LIN {X -0.212,Y -498.019,Z 383.978,A 0.000,B 0.000,C 90.000,E1 212.084} C_DIS
LIN {X 0.199,Y -493.119,Z 383.966,A 0.000,B 0.000,C 90.000,E1 209.922} C_DIS
LIN {X 0.159,Y -488.917,Z 383.956,A 0.000,B 0.000,C 90.000,E1 208.103} C_DIS
LIN {X 0.025,Y -484.697,Z 383.946,A 0.000,B 0.000,C 90.000,E1 206.283} C_DIS
LIN {X -0.193,Y -481.042,Z 383.938,A 0.000,B 0.000,C 90.000,E1 204.771} C_DIS
LIN {X -0.035,Y -477.293,Z 383.929,A 0.000,B 0.000,C 90.000,E1 203.206} C_DIS
LIN {X -0.131,Y -473.559,Z 383.920,A 0.000,B 0.000,C 90.000,E1 201.663} C_DIS
LIN {X 0.100,Y -469.164,Z 383.910,A 0.000,B 0.000,C 90.000,E1 199.758} C_DIS
LIN {X -0.148,Y -464.289,Z 383.898,A 0.000,B 0.000,C 90.000,E1 197.583} C_DIS
LIN {X -0.001,Y -460.326,Z 383.887,A 0.000,B 0.000,C 90.000,E1 195.662} C_DIS
LIN {X -0.193,Y -456.648,Z 383.876,A 0.000,B 0.000,C 90.000,E1 193.772} C_DIS
LIN {X 0.206,Y -453.691,Z 383.868,A 0.000,B 0.000,C 90.000,E1 192.119} C_DIS
LIN {X -0.131,Y -449.792,Z 383.855,A 0.000,B 0.000,C 90.000,E1 189.905} C_DIS
LIN {X 0.200,Y -447.685,Z 383.848,A 0.000,B 0.000,C 90.000,E1 188.568} C_DIS
LIN {X 0.012,Y -444.252,Z 383.835,A 0.000,B 0.000,C 90.000,E1 186.315} C_DIS
LIN {X 0.167,Y -439.679,Z 383.815,A 0.000,B 0.000,C 90.000,E1 182.694} C_DIS
LIN {X 0.131,Y -435.374,Z 383.786,A 0.000,B 0.000,C 90.000,E1 177.421} C_DIS
LIN {X -0.043,Y -433.968,Z 383.766,A 0.000,B 0.000,C 90.000,E1 173.799} C_DIS
LIN {X -0.105,Y -434.156,Z 383.740,A 0.000,B 0.000,C 90.000,E1 169.162} C_DIS
LIN {X -0.121,Y -435.862,Z 383.720,A 0.000,B 0.000,C 90.000,E1 165.519} C_DIS
LIN {X 0.098,Y -439.493,Z 383.698,A 0.000,B 0.000,C 90.000,E1 161.529} C_DIS
LIN {X -0.063,Y -444.442,Z 383.676,A 0.000,B 0.000,C 90.000,E1 157.614} C_DIS
LIN {X 0.018,Y -450.294,Z 383.656,A 0.000,B 0.000,C 90.000,E1 154.024} C_DIS
LIN {X 0.167,Y -457.487,Z 383.636,A 0.000,B 0.000,C 90.000,E1 150.461} C_DIS
LIN {X 0.284,Y -467.028,Z 383.615,A 0.000,B 0.000,C 90.000,E1 146.628} C_DIS
LIN {X -0.114,Y -471.651,Z 383.606,A 0.000,B 0.000,C 90.000,E1 145.102} C_DIS
LIN {X 0.087,Y -480.605,Z 383.591,A 0.000,B 0.000,C 90.000,E1 142.271} C_DIS
LIN {X -0.050,Y -486.857,Z 383.580,A 0.000,B 0.000,C 90.000,E1 140.436} C_DIS
LIN {X -0.269,Y -492.019,Z 383.572,A 0.000,B 0.000,C 90.000,E1 138.933} C_DIS
LIN {X 0.086,Y -496.064,Z 383.565,A 0.000,B 0.000,C 90.000,E1 137.676} C_DIS
LIN {X 0.008,Y -500.717,Z 383.557,A 0.000,B 0.000,C 90.000,E1 136.176} C_DIS
LIN {X 0.010,Y -505.000,Z 383.548,A 0.000,B 0.000,C 90.000,E1 134.676} C_DIS
LIN {X -0.026,Y -507.267,Z 383.543,A 0.000,B 0.000,C 90.000,E1 133.785} C_DIS
LIN {X -0.043,Y -509.313,Z 383.538,A 0.000,B 0.000,C 90.000,E1 132.894} C_DIS
LIN {X -0.009,Y -511.116,Z 383.533,A 0.000,B 0.000,C 90.000,E1 132.000} C_DIS
LIN {X -0.330,Y -512.746,Z 383.528,A 0.000,B 0.000,C 90.000,E1 131.148} C_DIS
LIN {X -0.166,Y -513.695,Z 383.525,A 0.000,B 0.000,C 90.000,E1 130.539} C_DIS
LIN {X -0.148,Y -515.089,Z 383.519,A 0.000,B 0.000,C 90.000,E1 129.358} C_DIS
LIN {X 0.032,Y -515.562,Z 383.515,A 0.000,B 0.000,C 90.000,E1 128.749} C_DIS
LIN {X -0.175,Y -515.754,Z 383.510,A 0.000,B 0.000,C 90.000,E1 127.890} C_DIS
LIN {X -0.067,Y -515.510,Z 383.506,A 0.000,B 0.000,C 90.000,E1 126.996} C_DIS
LIN {X 0.141,Y -514.805,Z 383.501,A 0.000,B 0.000,C 90.000,E1 126.091} C_DIS
LIN {X -0.002,Y -514.194,Z 383.497,A 0.000,B 0.000,C 90.000,E1 125.518} C_DIS
LIN {X 0.195,Y -512.974,Z 383.492,A 0.000,B 0.000,C 90.000,E1 124.612} C_DIS
LIN {X 0.035,Y -511.972,Z 383.489,A 0.000,B 0.000,C 90.000,E1 124.040} C_DIS
LIN {X -0.079,Y -510.194,Z 383.484,A 0.000,B 0.000,C 90.000,E1 123.166} C_DIS
LIN {X 0.125,Y -507.190,Z 383.478,A 0.000,B 0.000,C 90.000,E1 121.957} C_DIS
LIN {X -0.089,Y -505.513,Z 383.474,A 0.000,B 0.000,C 90.000,E1 121.386} C_DIS
LIN {X 0.164,Y -502.742,Z 383.469,A 0.000,B 0.000,C 90.000,E1 120.463} C_DIS
LIN {X -0.048,Y -499.626,Z 383.464,A 0.000,B 0.000,C 90.000,E1 119.589} C_DIS
LIN {X 0.174,Y -495.038,Z 383.458,A 0.000,B 0.000,C 90.000,E1 118.359} C_DIS
LIN {X -0.135,Y -490.540,Z 383.452,A 0.000,B 0.000,C 90.000,E1 117.334} C_DIS
LIN {X 0.156,Y -485.837,Z 383.446,A 0.000,B 0.000,C 90.000,E1 116.232} C_DIS
LIN {X -0.051,Y -481.546,Z 383.441,A 0.000,B 0.000,C 90.000,E1 115.335} C_DIS
LIN {X -0.121,Y -474.894,Z 383.433,A 0.000,B 0.000,C 90.000,E1 113.951} C_DIS
LIN {X 0.127,Y -467.905,Z 383.425,A 0.000,B 0.000,C 90.000,E1 112.514} C_DIS
LIN {X 0.070,Y -460.775,Z 383.417,A 0.000,B 0.000,C 90.000,E1 111.099} C_DIS
LIN {X 0.102,Y -456.211,Z 383.412,A 0.000,B 0.000,C 90.000,E1 110.174} C_DIS
LIN {X 0.063,Y -456.211,Z 383.412,A 0.000,B 0.000,C 90.000,E1 110.174} C_DIS
LIN {X -0.106,Y -457.519,Z 383.409,A 0.000,B 0.000,C 90.000,E1 109.685} C_DIS
LIN {X -0.161,Y -466.202,Z 383.386,A 0.000,B 0.000,C 90.000,E1 105.552} C_DIS
LIN {X 0.015,Y -467.767,Z 383.383,A 0.000,B 0.000,C 90.000,E1 104.898} C_DIS
LIN {X -0.013,Y -475.973,Z 383.357,A 0.000,B 0.000,C 90.000,E1 100.197} C_DIS
LIN {X 0.136,Y -476.681,Z 383.353,A 0.000,B 0.000,C 90.000,E1 99.557} C_DIS
LIN {X -0.218,Y -481.919,Z 383.331,A 0.000,B 0.000,C 90.000,E1 95.568} C_DIS
LIN {X 0.109,Y -482.204,Z 383.329,A 0.000,B 0.000,C 90.000,E1 95.220} C_DIS
LIN {X 0.048,Y -485.393,Z 383.305,A 0.000,B 0.000,C 90.000,E1 90.917} C_DIS
LIN {X -0.128,Y -485.529,Z 383.303,A 0.000,B 0.000,C 90.000,E1 90.630} C_DIS
LIN {X 0.080,Y -486.360,Z 383.281,A 0.000,B 0.000,C 90.000,E1 86.617} C_DIS
LIN {X -0.095,Y -486.368,Z 383.280,A 0.000,B 0.000,C 90.000,E1 86.331} C_DIS
LIN {X -0.106,Y -485.856,Z 383.275,A 0.000,B 0.000,C 90.000,E1 85.412} C_DIS
LIN {X -0.071,Y -484.692,Z 383.254,A 0.000,B 0.000,C 90.000,E1 81.724} C_DIS
LIN {X -0.203,Y -484.502,Z 383.252,A 0.000,B 0.000,C 90.000,E1 81.432} C_DIS
LIN {X 0.134,Y -480.434,Z 383.227,A 0.000,B 0.000,C 90.000,E1 76.769} C_DIS
LIN {X -0.225,Y -474.000,Z 383.200,A 0.000,B 0.000,C 90.000,E1 72.000} C_DIS
LIN {X 0.185,Y -473.730,Z 383.199,A 0.000,B 0.000,C 90.000,E1 71.819} C_DIS
LIN {X 0.144,Y -473.739,Z 383.199,A 0.000,B 0.000,C 90.000,E1 71.819} C_DIS
LIN {X 0.186,Y -482.818,Z 383.192,A 0.000,B 0.000,C 90.000,E1 70.550} C_DIS
LIN {X -0.179,Y -490.319,Z 383.186,A 0.000,B 0.000,C 90.000,E1 69.518} C_DIS
LIN {X -0.073,Y -496.699,Z 383.181,A 0.000,B 0.000,C 90.000,E1 68.592} C_DIS
LIN {X 0.110,Y -502.654,Z 383.176,A 0.000,B 0.000,C 90.000,E1 67.667} C_DIS
LIN {X 0.006,Y -510.529,Z 383.169,A 0.000,B 0.000,C 90.000,E1 66.357} C_DIS
LIN {X -0.302,Y -515.869,Z 383.163,A 0.000,B 0.000,C 90.000,E1 65.357} C_DIS
LIN {X -0.131,Y -517.950,Z 383.160,A 0.000,B 0.000,C 90.000,E1 64.897} C_DIS
LIN {X 0.171,Y -518.682,Z 383.160,A 0.000,B 0.000,C 90.000,E1 64.717} C_DIS
LIN {X 0.140,Y -520.608,Z 383.157,A 0.000,B 0.000,C 90.000,E1 64.280} C_DIS
LIN {X -0.189,Y -521.866,Z 383.156,A 0.000,B 0.000,C 90.000,E1 64.024} C_DIS
LIN {X -0.132,Y -524.336,Z 383.152,A 0.000,B 0.000,C 90.000,E1 63.435} C_DIS
LIN {X -0.294,Y -526.545,Z 383.149,A 0.000,B 0.000,C 90.000,E1 62.871} C_DIS
LIN {X -0.094,Y -530.547,Z 383.143,A 0.000,B 0.000,C 90.000,E1 61.691} C_DIS
LIN {X 0.205,Y -533.162,Z 383.138,A 0.000,B 0.000,C 90.000,E1 60.795} C_DIS
LIN {X 0.059,Y -535.621,Z 383.133,A 0.000,B 0.000,C 90.000,E1 59.950} C_DIS
LIN {X 0.204,Y -538.712,Z 383.127,A 0.000,B 0.000,C 90.000,E1 58.791} C_DIS
LIN {X 0.118,Y -541.438,Z 383.120,A 0.000,B 0.000,C 90.000,E1 57.661} C_DIS
LIN {X -0.098,Y -543.793,Z 383.114,A 0.000,B 0.000,C 90.000,E1 56.548} C_DIS
LIN {X 0.141,Y -545.326,Z 383.109,A 0.000,B 0.000,C 90.000,E1 55.674} C_DIS
LIN {X 0.213,Y -546.196,Z 383.106,A 0.000,B 0.000,C 90.000,E1 55.102} C_DIS
LIN {X -0.021,Y -546.950,Z 383.103,A 0.000,B 0.000,C 90.000,E1 54.562} C_DIS
LIN {X 0.111,Y -547.808,Z 383.098,A 0.000,B 0.000,C 90.000,E1 53.703} C_DIS
LIN {X 0.304,Y -548.476,Z 383.092,A 0.000,B 0.000,C 90.000,E1 52.557} C_DIS
LIN {X -0.029,Y -548.669,Z 383.089,A 0.000,B 0.000,C 90.000,E1 52.029} C_DIS
LIN {X 0.072,Y -548.643,Z 383.086,A 0.000,B 0.000,C 90.000,E1 51.457} C_DIS
LIN {X -0.205,Y -548.446,Z 383.081,A 0.000,B 0.000,C 90.000,E1 50.642} C_DIS
LIN {X 0.332,Y -547.697,Z 383.075,A 0.000,B 0.000,C 90.000,E1 49.461} C_DIS
LIN {X 0.039,Y -546.848,Z 383.070,A 0.000,B 0.000,C 90.000,E1 48.647} C_DIS
LIN {X -0.280,Y -545.318,Z 383.064,A 0.000,B 0.000,C 90.000,E1 47.553} C_DIS
LIN {X 0.165,Y -542.833,Z 383.055,A 0.000,B 0.000,C 90.000,E1 45.810} C_DIS
LIN {X 0.167,Y -540.290,Z 383.045,A 0.000,B 0.000,C 90.000,E1 44.109} C_DIS
LIN {X 0.100,Y -537.579,Z 383.034,A 0.000,B 0.000,C 90.000,E1 42.123} C_DIS
LIN {X -0.007,Y -534.998,Z 383.023,A 0.000,B 0.000,C 90.000,E1 40.135} C_DIS
LIN {X 0.300,Y -532.441,Z 383.012,A 0.000,B 0.000,C 90.000,E1 38.096} C_DIS
LIN {X 0.253,Y -530.574,Z 383.004,A 0.000,B 0.000,C 90.000,E1 36.664} C_DIS
LIN {X 0.149,Y -528.249,Z 382.994,A 0.000,B 0.000,C 90.000,E1 34.945} C_DIS
LIN {X 0.148,Y -526.357,Z 382.986,A 0.000,B 0.000,C 90.000,E1 33.499} C_DIS
LIN {X 0.187,Y -523.741,Z 382.975,A 0.000,B 0.000,C 90.000,E1 31.465} C_DIS
LIN {X 0.012,Y -520.809,Z 382.962,A 0.000,B 0.000,C 90.000,E1 29.155} C_DIS
LIN {X 0.165,Y -518.751,Z 382.952,A 0.000,B 0.000,C 90.000,E1 27.385} C_DIS
LIN {X 0.150,Y -516.488,Z 382.941,A 0.000,B 0.000,C 90.000,E1 25.335} C_DIS
LIN {X 0.115,Y -514.395,Z 382.929,A 0.000,B 0.000,C 90.000,E1 23.281} C_DIS
LIN {X -0.092,Y -511.838,Z 382.913,A 0.000,B 0.000,C 90.000,E1 20.355} C_DIS
LIN {X -0.094,Y -510.019,Z 382.898,A 0.000,B 0.000,C 90.000,E1 17.692} C_DIS
LIN {X -0.007,Y -508.836,Z 382.887,A 0.000,B 0.000,C 90.000,E1 15.607} C_DIS
LIN {X -0.052,Y -507.801,Z 382.872,A 0.000,B 0.000,C 90.000,E1 12.939} C_DIS
LIN {X -0.022,Y -507.332,Z 382.855,A 0.000,B 0.000,C 90.000,E1 9.962} C_DIS
LIN {X -0.122,Y -507.550,Z 382.841,A 0.000,B 0.000,C 90.000,E1 7.296} C_DIS
LIN {X -0.001,Y -508.745,Z 382.822,A 0.000,B 0.000,C 90.000,E1 4.012} C_DIS
LIN {X -0.043,Y -511.351,Z 382.803,A 0.000,B 0.000,C 90.000,E1 0.458} C_DIS
LIN {X -0.032,Y -515.651,Z 382.783,A 0.000,B 0.000,C 90.000,E1 356.846} C_DIS
LIN {X -0.032,Y -519.661,Z 382.768,A 0.000,B 0.000,C 90.000,E1 354.204} C_DIS
LIN {X -0.271,Y -523.319,Z 382.756,A 0.000,B 0.000,C 90.000,E1 352.186} C_DIS
LIN {X -0.151,Y -532.010,Z 382.734,A 0.000,B 0.000,C 90.000,E1 348.117} C_DIS
LIN {X 0.081,Y -539.526,Z 382.718,A 0.000,B 0.000,C 90.000,E1 345.227} C_DIS
LIN {X -0.263,Y -544.311,Z 382.709,A 0.000,B 0.000,C 90.000,E1 343.559} C_DIS
LIN {X 0.123,Y -546.738,Z 382.704,A 0.000,B 0.000,C 90.000,E1 342.670} C_DIS
LIN {X 0.000,Y -550.798,Z 382.696,A 0.000,B 0.000,C 90.000,E1 341.275} C_DIS
LIN {X -0.048,Y -554.954,Z 382.688,A 0.000,B 0.000,C 90.000,E1 339.880} C_DIS
LIN {X 0.172,Y -559.088,Z 382.681,A 0.000,B 0.000,C 90.000,E1 338.465} C_DIS
LIN {X -0.050,Y -563.189,Z 382.673,A 0.000,B 0.000,C 90.000,E1 337.102} C_DIS
LIN {X 0.123,Y -568.179,Z 382.664,A 0.000,B 0.000,C 90.000,E1 335.433} C_DIS
LIN {X -0.157,Y -573.249,Z 382.655,A 0.000,B 0.000,C 90.000,E1 333.819} C_DIS
LIN {X -0.235,Y -581.148,Z 382.641,A 0.000,B 0.000,C 90.000,E1 331.385} C_DIS
LIN {X 0.090,Y -588.403,Z 382.629,A 0.000,B 0.000,C 90.000,E1 329.203} C_DIS
LIN {X 0.117,Y -592.882,Z 382.622,A 0.000,B 0.000,C 90.000,E1 327.867} C_DIS
LIN {X 0.167,Y -599.167,Z 382.611,A 0.000,B 0.000,C 90.000,E1 326.008} C_DIS
LIN {X -0.125,Y -605.669,Z 382.601,A 0.000,B 0.000,C 90.000,E1 324.196} C_DIS
LIN {X 0.085,Y -612.260,Z 382.591,A 0.000,B 0.000,C 90.000,E1 322.351} C_DIS
LIN {X -0.271,Y -617.075,Z 382.584,A 0.000,B 0.000,C 90.000,E1 321.090} C_DIS
LIN {X -0.222,Y -622.892,Z 382.575,A 0.000,B 0.000,C 90.000,E1 319.542} C_DIS
LIN {X -0.127,Y -628.524,Z 382.567,A 0.000,B 0.000,C 90.000,E1 318.000} C_DIS
LIN {X -0.151,Y -632.208,Z 382.561,A 0.000,B 0.000,C 90.000,E1 316.986} C_DIS
LIN {X -0.126,Y -635.898,Z 382.555,A 0.000,B 0.000,C 90.000,E1 315.972} C_DIS
LIN {X 0.050,Y -643.196,Z 382.544,A 0.000,B 0.000,C 90.000,E1 313.947} C_DIS
LIN {X 0.090,Y -648.799,Z 382.536,A 0.000,B 0.000,C 90.000,E1 312.447} C_DIS
LIN {X 0.244,Y -655.166,Z 382.526,A 0.000,B 0.000,C 90.000,E1 310.701} C_DIS
LIN {X 0.125,Y -661.283,Z 382.517,A 0.000,B 0.000,C 90.000,E1 308.991} C_DIS
LIN {X 0.158,Y -666.149,Z 382.509,A 0.000,B 0.000,C 90.000,E1 307.523} C_DIS
LIN {X -0.219,Y -669.305,Z 382.503,A 0.000,B 0.000,C 90.000,E1 306.583} C_DIS
LIN {X -0.041,Y -673.071,Z 382.496,A 0.000,B 0.000,C 90.000,E1 305.358} C_DIS
LIN {X -0.043,Y -677.288,Z 382.488,A 0.000,B 0.000,C 90.000,E1 303.913} C_DIS
LIN {X -0.120,Y -679.965,Z 382.483,A 0.000,B 0.000,C 90.000,E1 302.959} C_DIS
LIN {X 0.226,Y -681.866,Z 382.479,A 0.000,B 0.000,C 90.000,E1 302.212} C_DIS
LIN {X -0.174,Y -684.909,Z 382.472,A 0.000,B 0.000,C 90.000,E1 301.052} C_DIS
LIN {X 0.244,Y -686.100,Z 382.470,A 0.000,B 0.000,C 90.000,E1 300.541} C_DIS
LIN {X -0.292,Y -687.664,Z 382.466,A 0.000,B 0.000,C 90.000,E1 299.873} C_DIS
LIN {X -0.219,Y -688.947,Z 382.462,A 0.000,B 0.000,C 90.000,E1 299.155} C_DIS
LIN {X -0.270,Y -690.464,Z 382.455,A 0.000,B 0.000,C 90.000,E1 297.975} C_DIS
LIN {X -0.170,Y -690.972,Z 382.451,A 0.000,B 0.000,C 90.000,E1 297.257} C_DIS
LIN {X -0.071,Y -691.259,Z 382.447,A 0.000,B 0.000,C 90.000,E1 296.539} C_DIS
LIN {X -0.278,Y -691.343,Z 382.444,A 0.000,B 0.000,C 90.000,E1 295.848} C_DIS
LIN {X -0.037,Y -691.243,Z 382.442,A 0.000,B 0.000,C 90.000,E1 295.591} C_DIS
LIN {X 0.202,Y -691.331,Z 382.441,A 0.000,B 0.000,C 90.000,E1 295.335} C_DIS
LIN {X -0.239,Y -691.030,Z 382.438,A 0.000,B 0.000,C 90.000,E1 294.899} C_DIS
LIN {X 0.190,Y -690.803,Z 382.434,A 0.000,B 0.000,C 90.000,E1 294.155} C_DIS
LIN {X -0.012,Y -690.231,Z 382.430,A 0.000,B 0.000,C 90.000,E1 293.462} C_DIS
LIN {X -0.223,Y -689.463,Z 382.426,A 0.000,B 0.000,C 90.000,E1 292.770} C_DIS
LIN {X 0.192,Y -688.369,Z 382.422,A 0.000,B 0.000,C 90.000,E1 292.025} C_DIS
LIN {X 0.092,Y -685.866,Z 382.415,A 0.000,B 0.000,C 90.000,E1 290.610} C_DIS
LIN {X -0.106,Y -682.586,Z 382.405,A 0.000,B 0.000,C 90.000,E1 288.960} C_DIS
LIN {X -0.081,Y -680.099,Z 382.399,A 0.000,B 0.000,C 90.000,E1 287.764} C_DIS
LIN {X -0.041,Y -678.147,Z 382.393,A 0.000,B 0.000,C 90.000,E1 286.804} C_DIS
LIN {X -0.179,Y -674.689,Z 382.384,A 0.000,B 0.000,C 90.000,E1 285.134} C_DIS
LIN {X -0.234,Y -669.113,Z 382.368,A 0.000,B 0.000,C 90.000,E1 282.243} C_DIS
LIN {X -0.046,Y -664.999,Z 382.353,A 0.000,B 0.000,C 90.000,E1 279.557} C_DIS
LIN {X -0.196,Y -660.985,Z 382.333,A 0.000,B 0.000,C 90.000,E1 275.910} C_DIS
LIN {X -0.128,Y -659.346,Z 382.318,A 0.000,B 0.000,C 90.000,E1 273.212} C_DIS
LIN {X 0.049,Y -658.757,Z 382.304,A 0.000,B 0.000,C 90.000,E1 270.745} C_DIS
LIN {X 0.073,Y -658.628,Z 382.295,A 0.000,B 0.000,C 90.000,E1 269.026} C_DIS
LIN {X 0.172,Y -658.705,Z 382.291,A 0.000,B 0.000,C 90.000,E1 268.282} C_DIS
LIN {X 0.047,Y -658.927,Z 382.280,A 0.000,B 0.000,C 90.000,E1 266.331} C_DIS
LIN {X 0.312,Y -659.082,Z 382.272,A 0.000,B 0.000,C 90.000,E1 264.837} C_DIS
LIN {X -0.212,Y -659.061,Z 382.267,A 0.000,B 0.000,C 90.000,E1 264.147} C_DIS
LIN {X -0.011,Y -658.779,Z 382.263,A 0.000,B 0.000,C 90.000,E1 263.394} C_DIS
LIN {X 0.112,Y -658.258,Z 382.259,A 0.000,B 0.000,C 90.000,E1 262.648} C_DIS
LIN {X 0.311,Y -657.608,Z 382.255,A 0.000,B 0.000,C 90.000,E1 261.894} C_DIS
LIN {X -0.145,Y -656.638,Z 382.251,A 0.000,B 0.000,C 90.000,E1 261.197} C_DIS
LIN {X -0.366,Y -656.173,Z 382.250,A 0.000,B 0.000,C 90.000,E1 260.971} C_DIS
LIN {X 0.041,Y -655.553,Z 382.247,A 0.000,B 0.000,C 90.000,E1 260.443} C_DIS
LIN {X 0.213,Y -654.345,Z 382.243,A 0.000,B 0.000,C 90.000,E1 259.690} C_DIS
LIN {X -0.275,Y -653.063,Z 382.239,A 0.000,B 0.000,C 90.000,E1 258.993} C_DIS
LIN {X -0.135,Y -651.333,Z 382.233,A 0.000,B 0.000,C 90.000,E1 257.993} C_DIS
LIN {X -0.008,Y -649.355,Z 382.228,A 0.000,B 0.000,C 90.000,E1 256.992} C_DIS
LIN {X 0.227,Y -647.739,Z 382.224,A 0.000,B 0.000,C 90.000,E1 256.228} C_DIS
LIN {X 0.301,Y -645.198,Z 382.218,A 0.000,B 0.000,C 90.000,E1 255.227} C_DIS
LIN {X -0.115,Y -642.407,Z 382.213,A 0.000,B 0.000,C 90.000,E1 254.267} C_DIS
LIN {X -0.103,Y -638.482,Z 382.206,A 0.000,B 0.000,C 90.000,E1 253.015} C_DIS
LIN {X -0.170,Y -634.126,Z 382.199,A 0.000,B 0.000,C 90.000,E1 251.764} C_DIS
LIN {X 0.078,Y -630.416,Z 382.193,A 0.000,B 0.000,C 90.000,E1 250.732} C_DIS
LIN {X 0.278,Y -625.534,Z 382.186,A 0.000,B 0.000,C 90.000,E1 249.444} C_DIS
LIN {X -0.174,Y -621.492,Z 382.180,A 0.000,B 0.000,C 90.000,E1 248.465} C_DIS
LIN {X -0.150,Y -615.178,Z 382.172,A 0.000,B 0.000,C 90.000,E1 246.922} C_DIS
LIN {X -0.062,Y -607.557,Z 382.162,A 0.000,B 0.000,C 90.000,E1 245.101} C_DIS
LIN {X 0.164,Y -600.939,Z 382.153,A 0.000,B 0.000,C 90.000,E1 243.512} C_DIS
LIN {X -0.287,Y -594.283,Z 382.144,A 0.000,B 0.000,C 90.000,E1 241.975} C_DIS
LIN {X 0.317,Y -588.841,Z 382.137,A 0.000,B 0.000,C 90.000,E1 240.589} C_DIS
LIN {X 0.217,Y -580.434,Z 382.125,A 0.000,B 0.000,C 90.000,E1 238.456} C_DIS
LIN {X 0.189,Y -572.528,Z 382.113,A 0.000,B 0.000,C 90.000,E1 236.294} C_DIS
LIN {X 0.220,Y -564.219,Z 382.099,A 0.000,B 0.000,C 90.000,E1 233.829} C_DIS
LIN {X -0.039,Y -559.593,Z 382.092,A 0.000,B 0.000,C 90.000,E1 232.477} C_DIS
LIN {X -0.039,Y -554.849,Z 382.084,A 0.000,B 0.000,C 90.000,E1 231.090} C_DIS
LIN {X 0.002,Y -546.340,Z 382.070,A 0.000,B 0.000,C 90.000,E1 228.566} C_DIS
LIN {X 0.061,Y -539.958,Z 382.059,A 0.000,B 0.000,C 90.000,E1 226.581} C_DIS
LIN {X -0.006,Y -534.551,Z 382.049,A 0.000,B 0.000,C 90.000,E1 224.879} C_DIS
LIN {X -0.157,Y -530.139,Z 382.041,A 0.000,B 0.000,C 90.000,E1 223.461} C_DIS
LIN {X 0.319,Y -524.906,Z 382.032,A 0.000,B 0.000,C 90.000,E1 221.676} C_DIS
LIN {X 0.272,Y -519.007,Z 382.020,A 0.000,B 0.000,C 90.000,E1 219.644} C_DIS
LIN {X 0.154,Y -513.317,Z 382.009,A 0.000,B 0.000,C 90.000,E1 217.604} C_DIS
LIN {X 0.202,Y -507.081,Z 381.996,A 0.000,B 0.000,C 90.000,E1 215.231} C_DIS
LIN {X 0.125,Y -502.630,Z 381.986,A 0.000,B 0.000,C 90.000,E1 213.452} C_DIS
LIN {X -0.044,Y -498.327,Z 381.976,A 0.000,B 0.000,C 90.000,E1 211.671} C_DIS
LIN {X -0.147,Y -494.179,Z 381.966,A 0.000,B 0.000,C 90.000,E1 209.873} C_DIS
LIN {X -0.173,Y -490.686,Z 381.957,A 0.000,B 0.000,C 90.000,E1 208.359} C_DIS
LIN {X -0.253,Y -485.788,Z 381.946,A 0.000,B 0.000,C 90.000,E1 206.232} C_DIS
LIN {X 0.197,Y -482.142,Z 381.937,A 0.000,B 0.000,C 90.000,E1 204.643} C_DIS
LIN {X -0.068,Y -478.405,Z 381.928,A 0.000,B 0.000,C 90.000,E1 203.131} C_DIS
LIN {X -0.129,Y -475.457,Z 381.922,A 0.000,B 0.000,C 90.000,E1 201.897} C_DIS
LIN {X -0.061,Y -470.317,Z 381.909,A 0.000,B 0.000,C 90.000,E1 199.704} C_DIS
LIN {X -0.067,Y -466.143,Z 381.899,A 0.000,B 0.000,C 90.000,E1 197.819} C_DIS
LIN {X -0.091,Y -461.496,Z 381.887,A 0.000,B 0.000,C 90.000,E1 195.607} C_DIS
LIN {X -0.035,Y -458.433,Z 381.878,A 0.000,B 0.000,C 90.000,E1 194.008} C_DIS
LIN {X -0.044,Y -455.447,Z 381.869,A 0.000,B 0.000,C 90.000,E1 192.411} C_DIS
LIN {X -0.129,Y -450.955,Z 381.855,A 0.000,B 0.000,C 90.000,E1 189.849} C_DIS
LIN {X 0.222,Y -448.835,Z 381.848,A 0.000,B 0.000,C 90.000,E1 188.511} C_DIS
LIN {X 0.067,Y -445.397,Z 381.835,A 0.000,B 0.000,C 90.000,E1 186.258} C_DIS
LIN {X -0.167,Y -440.791,Z 381.815,A 0.000,B 0.000,C 90.000,E1 182.694} C_DIS
LIN {X 0.101,Y -436.798,Z 381.789,A 0.000,B 0.000,C 90.000,E1 178.051} C_DIS
LIN {X -0.032,Y -435.628,Z 381.776,A 0.000,B 0.000,C 90.000,E1 175.755} C_DIS
LIN {X -0.129,Y -434.933,Z 381.764,A 0.000,B 0.000,C 90.000,E1 173.451} C_DIS
LIN {X 0.035,Y -435.111,Z 381.741,A 0.000,B 0.000,C 90.000,E1 169.454} C_DIS
LIN {X 0.189,Y -436.902,Z 381.719,A 0.000,B 0.000,C 90.000,E1 165.463} C_DIS
LIN {X 0.032,Y -440.529,Z 381.697,A 0.000,B 0.000,C 90.000,E1 161.529} C_DIS
LIN {X 0.229,Y -446.435,Z 381.672,A 0.000,B 0.000,C 90.000,E1 156.922} C_DIS
LIN {X -0.079,Y -451.905,Z 381.654,A 0.000,B 0.000,C 90.000,E1 153.717} C_DIS
LIN {X -0.273,Y -459.246,Z 381.634,A 0.000,B 0.000,C 90.000,E1 150.205} C_DIS
LIN {X -0.091,Y -469.012,Z 381.613,A 0.000,B 0.000,C 90.000,E1 146.373} C_DIS
LIN {X 0.195,Y -473.660,Z 381.604,A 0.000,B 0.000,C 90.000,E1 144.769} C_DIS
LIN {X -0.109,Y -481.755,Z 381.591,A 0.000,B 0.000,C 90.000,E1 142.316} C_DIS
LIN {X 0.164,Y -487.989,Z 381.580,A 0.000,B 0.000,C 90.000,E1 140.436} C_DIS
LIN {X -0.032,Y -493.150,Z 381.572,A 0.000,B 0.000,C 90.000,E1 138.933} C_DIS
LIN {X 0.007,Y -497.187,Z 381.565,A 0.000,B 0.000,C 90.000,E1 137.715} C_DIS
LIN {X -0.061,Y -501.831,Z 381.557,A 0.000,B 0.000,C 90.000,E1 136.215} C_DIS
LIN {X -0.047,Y -506.093,Z 381.548,A 0.000,B 0.000,C 90.000,E1 134.717} C_DIS
LIN {X 0.289,Y -508.341,Z 381.543,A 0.000,B 0.000,C 90.000,E1 133.785} C_DIS
LIN {X -0.062,Y -510.380,Z 381.539,A 0.000,B 0.000,C 90.000,E1 132.933} C_DIS
LIN {X -0.047,Y -512.170,Z 381.534,A 0.000,B 0.000,C 90.000,E1 132.043} C_DIS
LIN {X 0.110,Y -513.314,Z 381.530,A 0.000,B 0.000,C 90.000,E1 131.434} C_DIS
LIN {X 0.197,Y -514.738,Z 381.525,A 0.000,B 0.000,C 90.000,E1 130.539} C_DIS
LIN {X -0.168,Y -516.093,Z 381.519,A 0.000,B 0.000,C 90.000,E1 129.402} C_DIS
LIN {X -0.307,Y -516.536,Z 381.516,A 0.000,B 0.000,C 90.000,E1 128.830} C_DIS
LIN {X 0.223,Y -516.738,Z 381.511,A 0.000,B 0.000,C 90.000,E1 127.890} C_DIS
LIN {X 0.032,Y -516.522,Z 381.506,A 0.000,B 0.000,C 90.000,E1 127.030} C_DIS
LIN {X -0.161,Y -515.827,Z 381.501,A 0.000,B 0.000,C 90.000,E1 126.171} C_DIS
LIN {X 0.057,Y -514.841,Z 381.496,A 0.000,B 0.000,C 90.000,E1 125.264} C_DIS
LIN {X -0.083,Y -514.046,Z 381.493,A 0.000,B 0.000,C 90.000,E1 124.692} C_DIS
LIN {X 0.114,Y -512.497,Z 381.488,A 0.000,B 0.000,C 90.000,E1 123.785} C_DIS
LIN {X -0.053,Y -511.340,Z 381.485,A 0.000,B 0.000,C 90.000,E1 123.214} C_DIS
LIN {X 0.061,Y -507.652,Z 381.476,A 0.000,B 0.000,C 90.000,E1 121.720} C_DIS
LIN {X -0.097,Y -504.977,Z 381.471,A 0.000,B 0.000,C 90.000,E1 120.846} C_DIS
LIN {X -0.160,Y -503.089,Z 381.468,A 0.000,B 0.000,C 90.000,E1 120.256} C_DIS
LIN {X -0.232,Y -501.032,Z 381.465,A 0.000,B 0.000,C 90.000,E1 119.667} C_DIS
LIN {X 0.017,Y -496.485,Z 381.458,A 0.000,B 0.000,C 90.000,E1 118.437} C_DIS
LIN {X 0.163,Y -492.805,Z 381.453,A 0.000,B 0.000,C 90.000,E1 117.513} C_DIS
LIN {X 0.057,Y -486.854,Z 381.445,A 0.000,B 0.000,C 90.000,E1 116.155} C_DIS
LIN {X 0.294,Y -482.619,Z 381.440,A 0.000,B 0.000,C 90.000,E1 115.207} C_DIS
LIN {X 0.238,Y -476.008,Z 381.433,A 0.000,B 0.000,C 90.000,E1 113.823} C_DIS
LIN {X -0.076,Y -470.637,Z 381.426,A 0.000,B 0.000,C 90.000,E1 112.770} C_DIS
LIN {X -0.077,Y -463.586,Z 381.419,A 0.000,B 0.000,C 90.000,E1 111.354} C_DIS
LIN {X -0.111,Y -456.818,Z 381.411,A 0.000,B 0.000,C 90.000,E1 109.993} C_DIS
LIN {X -0.151,Y -456.797,Z 381.411,A 0.000,B 0.000,C 90.000,E1 109.993} C_DIS
LIN {X -0.029,Y -457.371,Z 381.410,A 0.000,B 0.000,C 90.000,E1 109.758} C_DIS
LIN {X 0.056,Y -466.003,Z 381.387,A 0.000,B 0.000,C 90.000,E1 105.607} C_DIS
LIN {X -0.221,Y -467.570,Z 381.383,A 0.000,B 0.000,C 90.000,E1 105.009} C_DIS
LIN {X -0.038,Y -468.578,Z 381.380,A 0.000,B 0.000,C 90.000,E1 104.356} C_DIS
LIN {X 0.190,Y -475.803,Z 381.357,A 0.000,B 0.000,C 90.000,E1 100.254} C_DIS
LIN {X 0.028,Y -476.306,Z 381.355,A 0.000,B 0.000,C 90.000,E1 99.962} C_DIS
LIN {X -0.025,Y -481.790,Z 381.331,A 0.000,B 0.000,C 90.000,E1 95.625} C_DIS
LIN {X -0.178,Y -482.172,Z 381.330,A 0.000,B 0.000,C 90.000,E1 95.334} C_DIS
LIN {X 0.236,Y -485.308,Z 381.306,A 0.000,B 0.000,C 90.000,E1 90.974} C_DIS
LIN {X 0.061,Y -485.537,Z 381.304,A 0.000,B 0.000,C 90.000,E1 90.688} C_DIS
LIN {X -0.217,Y -486.320,Z 381.282,A 0.000,B 0.000,C 90.000,E1 86.731} C_DIS
LIN {X -0.082,Y -486.304,Z 381.278,A 0.000,B 0.000,C 90.000,E1 86.102} C_DIS
LIN {X 0.123,Y -484.695,Z 381.254,A 0.000,B 0.000,C 90.000,E1 81.781} C_DIS
LIN {X -0.009,Y -484.599,Z 381.253,A 0.000,B 0.000,C 90.000,E1 81.489} C_DIS
LIN {X -0.130,Y -480.533,Z 381.227,A 0.000,B 0.000,C 90.000,E1 76.881} C_DIS
LIN {X 0.081,Y -474.065,Z 381.200,A 0.000,B 0.000,C 90.000,E1 72.000} C_DIS
LIN {X 0.040,Y -474.082,Z 381.200,A 0.000,B 0.000,C 90.000,E1 72.000} C_DIS
LIN {X 0.201,Y -482.648,Z 381.193,A 0.000,B 0.000,C 90.000,E1 70.786} C_DIS
LIN {X 0.056,Y -489.024,Z 381.188,A 0.000,B 0.000,C 90.000,E1 69.880} C_DIS
LIN {X -0.240,Y -498.118,Z 381.181,A 0.000,B 0.000,C 90.000,E1 68.592} C_DIS
LIN {X 0.153,Y -502.931,Z 381.177,A 0.000,B 0.000,C 90.000,E1 67.794} C_DIS
LIN {X 0.035,Y -509.893,Z 381.170,A 0.000,B 0.000,C 90.000,E1 66.613} C_DIS
LIN {X 0.068,Y -513.713,Z 381.166,A 0.000,B 0.000,C 90.000,E1 65.869} C_DIS
LIN {X 0.054,Y -516.573,Z 381.163,A 0.000,B 0.000,C 90.000,E1 65.281} C_DIS
LIN {X -0.154,Y -519.199,Z 381.159,A 0.000,B 0.000,C 90.000,E1 64.717} C_DIS
LIN {X -0.183,Y -520.990,Z 381.157,A 0.000,B 0.000,C 90.000,E1 64.280} C_DIS
LIN {X 0.120,Y -521.669,Z 381.156,A 0.000,B 0.000,C 90.000,E1 64.101} C_DIS
LIN {X -0.136,Y -523.306,Z 381.154,A 0.000,B 0.000,C 90.000,E1 63.691} C_DIS
LIN {X 0.172,Y -523.953,Z 381.153,A 0.000,B 0.000,C 90.000,E1 63.512} C_DIS
LIN {X 0.092,Y -528.065,Z 381.147,A 0.000,B 0.000,C 90.000,E1 62.359} C_DIS
LIN {X -0.106,Y -530.902,Z 381.142,A 0.000,B 0.000,C 90.000,E1 61.513} C_DIS
LIN {X -0.130,Y -535.018,Z 381.134,A 0.000,B 0.000,C 90.000,E1 60.078} C_DIS
LIN {X 0.006,Y -538.147,Z 381.127,A 0.000,B 0.000,C 90.000,E1 58.918} C_DIS
LIN {X -0.075,Y -541.570,Z 381.119,A 0.000,B 0.000,C 90.000,E1 57.502} C_DIS
LIN {X -0.131,Y -543.965,Z 381.113,A 0.000,B 0.000,C 90.000,E1 56.373} C_DIS
LIN {X -0.038,Y -545.544,Z 381.108,A 0.000,B 0.000,C 90.000,E1 55.515} C_DIS
LIN {X -0.236,Y -546.838,Z 381.104,A 0.000,B 0.000,C 90.000,E1 54.689} C_DIS
LIN {X -0.148,Y -547.537,Z 381.101,A 0.000,B 0.000,C 90.000,E1 54.116} C_DIS
LIN {X -0.055,Y -548.169,Z 381.097,A 0.000,B 0.000,C 90.000,E1 53.543} C_DIS
LIN {X 0.148,Y -548.965,Z 381.091,A 0.000,B 0.000,C 90.000,E1 52.396} C_DIS
LIN {X 0.305,Y -549.206,Z 381.087,A 0.000,B 0.000,C 90.000,E1 51.537} C_DIS
LIN {X 0.031,Y -549.197,Z 381.082,A 0.000,B 0.000,C 90.000,E1 50.723} C_DIS
LIN {X -0.194,Y -548.571,Z 381.076,A 0.000,B 0.000,C 90.000,E1 49.622} C_DIS
LIN {X -0.077,Y -547.551,Z 381.069,A 0.000,B 0.000,C 90.000,E1 48.485} C_DIS
LIN {X 0.018,Y -546.005,Z 381.063,A 0.000,B 0.000,C 90.000,E1 47.349} C_DIS
LIN {X 0.079,Y -543.541,Z 381.054,A 0.000,B 0.000,C 90.000,E1 45.648} C_DIS
LIN {X -0.289,Y -540.642,Z 381.043,A 0.000,B 0.000,C 90.000,E1 43.704} C_DIS
LIN {X 0.047,Y -538.309,Z 381.033,A 0.000,B 0.000,C 90.000,E1 41.962} C_DIS
LIN {X 0.020,Y -535.748,Z 381.022,A 0.000,B 0.000,C 90.000,E1 39.967} C_DIS
LIN {X -0.052,Y -533.169,Z 381.011,A 0.000,B 0.000,C 90.000,E1 37.971} C_DIS
LIN {X 0.237,Y -531.293,Z 381.003,A 0.000,B 0.000,C 90.000,E1 36.503} C_DIS
LIN {X -0.142,Y -529.376,Z 380.995,A 0.000,B 0.000,C 90.000,E1 35.105} C_DIS
LIN {X -0.114,Y -527.483,Z 380.987,A 0.000,B 0.000,C 90.000,E1 33.658} C_DIS
LIN {X 0.240,Y -524.892,Z 380.976,A 0.000,B 0.000,C 90.000,E1 31.592} C_DIS
LIN {X 0.094,Y -521.969,Z 380.963,A 0.000,B 0.000,C 90.000,E1 29.283} C_DIS
LIN {X -0.055,Y -519.574,Z 380.951,A 0.000,B 0.000,C 90.000,E1 27.257} C_DIS
LIN {X -0.049,Y -517.344,Z 380.940,A 0.000,B 0.000,C 90.000,E1 25.207} C_DIS
LIN {X 0.141,Y -515.276,Z 380.929,A 0.000,B 0.000,C 90.000,E1 23.131} C_DIS
LIN {X 0.121,Y -512.977,Z 380.914,A 0.000,B 0.000,C 90.000,E1 20.482} C_DIS
LIN {X 0.268,Y -510.973,Z 380.897,A 0.000,B 0.000,C 90.000,E1 17.511} C_DIS
LIN {X -0.157,Y -509.688,Z 380.884,A 0.000,B 0.000,C 90.000,E1 15.190} C_DIS
LIN {X -0.249,Y -508.861,Z 380.871,A 0.000,B 0.000,C 90.000,E1 12.827} C_DIS
LIN {X -0.168,Y -508.469,Z 380.855,A 0.000,B 0.000,C 90.000,E1 9.849} C_DIS
LIN {X 0.232,Y -508.811,Z 380.838,A 0.000,B 0.000,C 90.000,E1 6.834} C_DIS
LIN {X -0.047,Y -510.018,Z 380.822,A 0.000,B 0.000,C 90.000,E1 3.898} C_DIS
LIN {X 0.135,Y -512.176,Z 380.805,A 0.000,B 0.000,C 90.000,E1 0.917} C_DIS
LIN {X 0.058,Y -516.530,Z 380.784,A 0.000,B 0.000,C 90.000,E1 357.135} C_DIS
LIN {X 0.124,Y -520.528,Z 380.770,A 0.000,B 0.000,C 90.000,E1 354.489} C_DIS
LIN {X -0.134,Y -525.203,Z 380.755,A 0.000,B 0.000,C 90.000,E1 351.894} C_DIS
LIN {X 0.094,Y -534.115,Z 380.732,A 0.000,B 0.000,C 90.000,E1 347.825} C_DIS
LIN {X -0.186,Y -540.978,Z 380.718,A 0.000,B 0.000,C 90.000,E1 345.283} C_DIS
LIN {X -0.205,Y -544.986,Z 380.710,A 0.000,B 0.000,C 90.000,E1 343.866} C_DIS
LIN {X -0.280,Y -549.884,Z 380.701,A 0.000,B 0.000,C 90.000,E1 342.181} C_DIS
LIN {X -0.095,Y -553.168,Z 380.695,A 0.000,B 0.000,C 90.000,E1 341.040} C_DIS
LIN {X 0.087,Y -557.296,Z 380.687,A 0.000,B 0.000,C 90.000,E1 339.625} C_DIS
LIN {X -0.156,Y -560.655,Z 380.681,A 0.000,B 0.000,C 90.000,E1 338.539} C_DIS
LIN {X -0.141,Y -564.804,Z 380.673,A 0.000,B 0.000,C 90.000,E1 337.155} C_DIS
LIN {X 0.072,Y -569.749,Z 380.664,A 0.000,B 0.000,C 90.000,E1 335.485} C_DIS
LIN {X 0.093,Y -574.800,Z 380.655,A 0.000,B 0.000,C 90.000,E1 333.845} C_DIS
LIN {X -0.050,Y -581.813,Z 380.643,A 0.000,B 0.000,C 90.000,E1 331.691} C_DIS
LIN {X 0.132,Y -588.070,Z 380.632,A 0.000,B 0.000,C 90.000,E1 329.793} C_DIS
LIN {X -0.036,Y -591.728,Z 380.626,A 0.000,B 0.000,C 90.000,E1 328.742} C_DIS
LIN {X 0.044,Y -596.213,Z 380.619,A 0.000,B 0.000,C 90.000,E1 327.406} C_DIS
LIN {X -0.331,Y -602.530,Z 380.609,A 0.000,B 0.000,C 90.000,E1 325.595} C_DIS
LIN {X 0.027,Y -608.162,Z 380.600,A 0.000,B 0.000,C 90.000,E1 323.989} C_DIS
LIN {X -0.190,Y -614.791,Z 380.590,A 0.000,B 0.000,C 90.000,E1 322.190} C_DIS
LIN {X -0.331,Y -618.658,Z 380.584,A 0.000,B 0.000,C 90.000,E1 321.170} C_DIS
LIN {X 0.300,Y -623.504,Z 380.577,A 0.000,B 0.000,C 90.000,E1 319.828} C_DIS
LIN {X -0.001,Y -629.193,Z 380.569,A 0.000,B 0.000,C 90.000,E1 318.324} C_DIS
LIN {X -0.130,Y -633.776,Z 380.561,A 0.000,B 0.000,C 90.000,E1 317.067} C_DIS
LIN {X -0.182,Y -638.343,Z 380.554,A 0.000,B 0.000,C 90.000,E1 315.810} C_DIS
LIN {X 0.061,Y -645.706,Z 380.543,A 0.000,B 0.000,C 90.000,E1 313.785} C_DIS
LIN {X 0.208,Y -650.329,Z 380.536,A 0.000,B 0.000,C 90.000,E1 312.528} C_DIS
LIN {X -0.052,Y -655.778,Z 380.528,A 0.000,B 0.000,C 90.000,E1 311.067} C_DIS
LIN {X -0.107,Y -658.482,Z 380.524,A 0.000,B 0.000,C 90.000,E1 310.334} C_DIS
LIN {X -0.195,Y -662.817,Z 380.517,A 0.000,B 0.000,C 90.000,E1 309.116} C_DIS
LIN {X -0.141,Y -667.682,Z 380.509,A 0.000,B 0.000,C 90.000,E1 307.649} C_DIS
LIN {X 0.014,Y -671.605,Z 380.502,A 0.000,B 0.000,C 90.000,E1 306.423} C_DIS
LIN {X 0.241,Y -674.575,Z 380.497,A 0.000,B 0.000,C 90.000,E1 305.438} C_DIS
LIN {X -0.166,Y -675.329,Z 380.496,A 0.000,B 0.000,C 90.000,E1 305.231} C_DIS
LIN {X -0.120,Y -679.428,Z 380.488,A 0.000,B 0.000,C 90.000,E1 303.785} C_DIS
LIN {X 0.221,Y -681.395,Z 380.484,A 0.000,B 0.000,C 90.000,E1 303.038} C_DIS
LIN {X 0.008,Y -683.226,Z 380.480,A 0.000,B 0.000,C 90.000,E1 302.339} C_DIS
LIN {X -0.178,Y -684.363,Z 380.477,A 0.000,B 0.000,C 90.000,E1 301.878} C_DIS
LIN {X 0.004,Y -685.536,Z 380.474,A 0.000,B 0.000,C 90.000,E1 301.386} C_DIS
LIN {X 0.047,Y -687.229,Z 380.470,A 0.000,B 0.000,C 90.000,E1 300.669} C_DIS
LIN {X 0.117,Y -688.693,Z 380.466,A 0.000,B 0.000,C 90.000,E1 299.951} C_DIS
LIN {X -0.399,Y -689.859,Z 380.463,A 0.000,B 0.000,C 90.000,E1 299.283} C_DIS
LIN {X -0.066,Y -690.927,Z 380.457,A 0.000,B 0.000,C 90.000,E1 298.309} C_DIS
LIN {X -0.198,Y -691.416,Z 380.455,A 0.000,B 0.000,C 90.000,E1 297.847} C_DIS
LIN {X -0.088,Y -691.831,Z 380.451,A 0.000,B 0.000,C 90.000,E1 297.129} C_DIS
LIN {X -0.223,Y -691.986,Z 380.448,A 0.000,B 0.000,C 90.000,E1 296.668} C_DIS
LIN {X 0.200,Y -691.858,Z 380.444,A 0.000,B 0.000,C 90.000,E1 295.924} C_DIS
LIN {X 0.302,Y -691.560,Z 380.440,A 0.000,B 0.000,C 90.000,E1 295.207} C_DIS
LIN {X -0.338,Y -690.674,Z 380.434,A 0.000,B 0.000,C 90.000,E1 294.079} C_DIS
LIN {X 0.131,Y -690.175,Z 380.431,A 0.000,B 0.000,C 90.000,E1 293.567} C_DIS
LIN {X 0.097,Y -688.529,Z 380.424,A 0.000,B 0.000,C 90.000,E1 292.386} C_DIS
LIN {X -0.217,Y -686.398,Z 380.418,A 0.000,B 0.000,C 90.000,E1 291.227} C_DIS
LIN {X 0.162,Y -685.013,Z 380.414,A 0.000,B 0.000,C 90.000,E1 290.482} C_DIS
LIN {X -0.243,Y -682.191,Z 380.406,A 0.000,B 0.000,C 90.000,E1 289.087} C_DIS
LIN {X -0.011,Y -679.571,Z 380.399,A 0.000,B 0.000,C 90.000,E1 287.873} C_DIS
LIN {X 0.015,Y -677.551,Z 380.394,A 0.000,B 0.000,C 90.000,E1 286.913} C_DIS
LIN {X -0.203,Y -673.508,Z 380.383,A 0.000,B 0.000,C 90.000,E1 285.009} C_DIS
LIN {X 0.332,Y -667.932,Z 380.367,A 0.000,B 0.000,C 90.000,E1 282.063} C_DIS
LIN {X -0.194,Y -663.865,Z 380.352,A 0.000,B 0.000,C 90.000,E1 279.434} C_DIS
LIN {X -0.175,Y -660.321,Z 380.335,A 0.000,B 0.000,C 90.000,E1 276.258} C_DIS
LIN {X -0.270,Y -658.457,Z 380.318,A 0.000,B 0.000,C 90.000,E1 273.326} C_DIS
LIN {X -0.310,Y -657.799,Z 380.303,A 0.000,B 0.000,C 90.000,E1 270.630} C_DIS
LIN {X -0.198,Y -657.828,Z 380.290,A 0.000,B 0.000,C 90.000,E1 268.165} C_DIS
LIN {X -0.176,Y -658.181,Z 380.280,A 0.000,B 0.000,C 90.000,E1 266.445} C_DIS
LIN {X 0.273,Y -658.463,Z 380.273,A 0.000,B 0.000,C 90.000,E1 265.179} C_DIS
LIN {X -0.253,Y -658.524,Z 380.269,A 0.000,B 0.000,C 90.000,E1 264.489} C_DIS
LIN {X -0.125,Y -658.371,Z 380.265,A 0.000,B 0.000,C 90.000,E1 263.742} C_DIS
LIN {X -0.007,Y -658.084,Z 380.261,A 0.000,B 0.000,C 90.000,E1 262.996} C_DIS
LIN {X -0.150,Y -657.201,Z 380.254,A 0.000,B 0.000,C 90.000,E1 261.781} C_DIS
LIN {X -0.270,Y -656.871,Z 380.253,A 0.000,B 0.000,C 90.000,E1 261.546} C_DIS
LIN {X 0.285,Y -656.743,Z 380.252,A 0.000,B 0.000,C 90.000,E1 261.254} C_DIS
LIN {X 0.064,Y -656.317,Z 380.250,A 0.000,B 0.000,C 90.000,E1 261.027} C_DIS
LIN {X -0.176,Y -655.816,Z 380.247,A 0.000,B 0.000,C 90.000,E1 260.557} C_DIS
LIN {X 0.003,Y -654.794,Z 380.243,A 0.000,B 0.000,C 90.000,E1 259.803} C_DIS
LIN {X -0.080,Y -652.914,Z 380.237,A 0.000,B 0.000,C 90.000,E1 258.578} C_DIS
LIN {X -0.073,Y -651.246,Z 380.231,A 0.000,B 0.000,C 90.000,E1 257.589} C_DIS
LIN {X 0.046,Y -649.313,Z 380.226,A 0.000,B 0.000,C 90.000,E1 256.589} C_DIS
LIN {X -0.352,Y -647.646,Z 380.221,A 0.000,B 0.000,C 90.000,E1 255.880} C_DIS
LIN {X -0.117,Y -645.155,Z 380.216,A 0.000,B 0.000,C 90.000,E1 254.866} C_DIS
LIN {X 0.065,Y -643.098,Z 380.212,A 0.000,B 0.000,C 90.000,E1 254.102} C_DIS
LIN {X 0.238,Y -640.035,Z 380.206,A 0.000,B 0.000,C 90.000,E1 253.087} C_DIS
LIN {X -0.218,Y -635.792,Z 380.199,A 0.000,B 0.000,C 90.000,E1 251.873} C_DIS
LIN {X 0.041,Y -633.111,Z 380.195,A 0.000,B 0.000,C 90.000,E1 251.094} C_DIS
LIN {X 0.277,Y -629.297,Z 380.189,A 0.000,B 0.000,C 90.000,E1 250.061} C_DIS
LIN {X -0.130,Y -625.381,Z 380.184,A 0.000,B 0.000,C 90.000,E1 249.082} C_DIS
LIN {X -0.017,Y -620.243,Z 380.177,A 0.000,B 0.000,C 90.000,E1 247.794} C_DIS
LIN {X -0.306,Y -615.993,Z 380.171,A 0.000,B 0.000,C 90.000,E1 246.794} C_DIS
LIN {X -0.156,Y -609.486,Z 380.162,A 0.000,B 0.000,C 90.000,E1 245.229} C_DIS
LIN {X 0.111,Y -602.905,Z 380.154,A 0.000,B 0.000,C 90.000,E1 243.640} C_DIS
LIN {X -0.221,Y -597.389,Z 380.146,A 0.000,B 0.000,C 90.000,E1 242.359} C_DIS
LIN {X 0.341,Y -590.852,Z 380.138,A 0.000,B 0.000,C 90.000,E1 240.717} C_DIS
LIN {X 0.163,Y -581.396,Z 380.124,A 0.000,B 0.000,C 90.000,E1 238.329} C_DIS
LIN {X 0.156,Y -573.546,Z 380.112,A 0.000,B 0.000,C 90.000,E1 236.167} C_DIS
LIN {X -0.027,Y -567.034,Z 380.102,A 0.000,B 0.000,C 90.000,E1 234.276} C_DIS
LIN {X -0.011,Y -563.433,Z 380.095,A 0.000,B 0.000,C 90.000,E1 233.176} C_DIS
LIN {X -0.282,Y -558.746,Z 380.088,A 0.000,B 0.000,C 90.000,E1 231.823} C_DIS
LIN {X -0.297,Y -553.936,Z 380.080,A 0.000,B 0.000,C 90.000,E1 230.436} C_DIS
LIN {X -0.007,Y -547.378,Z 380.069,A 0.000,B 0.000,C 90.000,E1 228.447} C_DIS
LIN {X 0.102,Y -541.897,Z 380.060,A 0.000,B 0.000,C 90.000,E1 226.743} C_DIS
LIN {X 0.090,Y -537.391,Z 380.052,A 0.000,B 0.000,C 90.000,E1 225.324} C_DIS
LIN {X -0.041,Y -532.089,Z 380.042,A 0.000,B 0.000,C 90.000,E1 223.623} C_DIS
LIN {X 0.050,Y -525.927,Z 380.031,A 0.000,B 0.000,C 90.000,E1 221.595} C_DIS
LIN {X 0.031,Y -520.031,Z 380.020,A 0.000,B 0.000,C 90.000,E1 219.564} C_DIS
LIN {X -0.061,Y -514.343,Z 380.008,A 0.000,B 0.000,C 90.000,E1 217.523} C_DIS
LIN {X 0.015,Y -508.110,Z 379.995,A 0.000,B 0.000,C 90.000,E1 215.152} C_DIS
LIN {X -0.154,Y -502.934,Z 379.984,A 0.000,B 0.000,C 90.000,E1 213.086} C_DIS
LIN {X -0.295,Y -497.981,Z 379.972,A 0.000,B 0.000,C 90.000,E1 211.003} C_DIS
LIN {X 0.025,Y -493.828,Z 379.962,A 0.000,B 0.000,C 90.000,E1 209.155} C_DIS
LIN {X 0.011,Y -489.636,Z 379.952,A 0.000,B 0.000,C 90.000,E1 207.334} C_DIS
LIN {X 0.090,Y -486.853,Z 379.945,A 0.000,B 0.000,C 90.000,E1 206.104} C_DIS
LIN {X -0.082,Y -483.251,Z 379.937,A 0.000,B 0.000,C 90.000,E1 204.591} C_DIS
LIN {X 0.122,Y -479.526,Z 379.928,A 0.000,B 0.000,C 90.000,E1 203.025} C_DIS
LIN {X 0.085,Y -476.586,Z 379.921,A 0.000,B 0.000,C 90.000,E1 201.791} C_DIS
LIN {X -0.092,Y -471.462,Z 379.909,A 0.000,B 0.000,C 90.000,E1 199.631} C_DIS
LIN {X -0.224,Y -467.271,Z 379.899,A 0.000,B 0.000,C 90.000,E1 197.764} C_DIS
LIN {X -0.006,Y -463.318,Z 379.888,A 0.000,B 0.000,C 90.000,E1 195.843} C_DIS
LIN {X 0.214,Y -458.981,Z 379.876,A 0.000,B 0.000,C 90.000,E1 193.592} C_DIS
LIN {X -0.111,Y -456.609,Z 379.869,A 0.000,B 0.000,C 90.000,E1 192.355} C_DIS
LIN {X -0.155,Y -452.132,Z 379.854,A 0.000,B 0.000,C 90.000,E1 189.792} C_DIS
LIN {X -0.151,Y -448.484,Z 379.842,A 0.000,B 0.000,C 90.000,E1 187.530} C_DIS
LIN {X -0.183,Y -444.725,Z 379.827,A 0.000,B 0.000,C 90.000,E1 184.935} C_DIS
LIN {X -0.029,Y -440.523,Z 379.807,A 0.000,B 0.000,C 90.000,E1 181.318} C_DIS
LIN {X 0.119,Y -437.361,Z 379.784,A 0.000,B 0.000,C 90.000,E1 177.020} C_DIS
LIN {X -0.065,Y -436.148,Z 379.765,A 0.000,B 0.000,C 90.000,E1 173.742} C_DIS
LIN {X -0.014,Y -436.267,Z 379.740,A 0.000,B 0.000,C 90.000,E1 169.106} C_DIS
LIN {X 0.055,Y -437.944,Z 379.719,A 0.000,B 0.000,C 90.000,E1 165.463} C_DIS
LIN {X 0.088,Y -441.546,Z 379.697,A 0.000,B 0.000,C 90.000,E1 161.511} C_DIS
LIN {X -0.080,Y -446.979,Z 379.674,A 0.000,B 0.000,C 90.000,E1 157.283} C_DIS
LIN {X 0.171,Y -451.766,Z 379.658,A 0.000,B 0.000,C 90.000,E1 154.332} C_DIS
LIN {X 0.177,Y -457.446,Z 379.641,A 0.000,B 0.000,C 90.000,E1 151.435} C_DIS
LIN {X -0.047,Y -467.473,Z 379.618,A 0.000,B 0.000,C 90.000,E1 147.327} C_DIS
LIN {X 0.078,Y -477.705,Z 379.599,A 0.000,B 0.000,C 90.000,E1 143.863} C_DIS
LIN {X -0.129,Y -483.895,Z 379.589,A 0.000,B 0.000,C 90.000,E1 142.029} C_DIS
LIN {X -0.188,Y -490.126,Z 379.579,A 0.000,B 0.000,C 90.000,E1 140.194} C_DIS
LIN {X 0.184,Y -494.255,Z 379.572,A 0.000,B 0.000,C 90.000,E1 138.933} C_DIS
LIN {X -0.127,Y -498.268,Z 379.565,A 0.000,B 0.000,C 90.000,E1 137.757} C_DIS
LIN {X 0.197,Y -502.899,Z 379.557,A 0.000,B 0.000,C 90.000,E1 136.215} C_DIS
LIN {X 0.006,Y -506.303,Z 379.550,A 0.000,B 0.000,C 90.000,E1 135.040} C_DIS
LIN {X -0.021,Y -508.646,Z 379.545,A 0.000,B 0.000,C 90.000,E1 134.150} C_DIS
LIN {X 0.244,Y -511.382,Z 379.539,A 0.000,B 0.000,C 90.000,E1 132.933} C_DIS
LIN {X 0.019,Y -512.616,Z 379.535,A 0.000,B 0.000,C 90.000,E1 132.366} C_DIS
LIN {X 0.096,Y -514.253,Z 379.531,A 0.000,B 0.000,C 90.000,E1 131.472} C_DIS
LIN {X -0.193,Y -515.649,Z 379.526,A 0.000,B 0.000,C 90.000,E1 130.620} C_DIS
LIN {X -0.144,Y -516.946,Z 379.519,A 0.000,B 0.000,C 90.000,E1 129.439} C_DIS
LIN {X 0.051,Y -517.341,Z 379.516,A 0.000,B 0.000,C 90.000,E1 128.830} C_DIS
LIN {X -0.075,Y -517.494,Z 379.513,A 0.000,B 0.000,C 90.000,E1 128.257} C_DIS
LIN {X -0.006,Y -517.234,Z 379.506,A 0.000,B 0.000,C 90.000,E1 127.076} C_DIS
LIN {X -0.195,Y -516.553,Z 379.501,A 0.000,B 0.000,C 90.000,E1 126.217} C_DIS
LIN {X 0.026,Y -515.563,Z 379.496,A 0.000,B 0.000,C 90.000,E1 125.311} C_DIS
LIN {X -0.112,Y -514.757,Z 379.493,A 0.000,B 0.000,C 90.000,E1 124.739} C_DIS
LIN {X 0.088,Y -513.252,Z 379.488,A 0.000,B 0.000,C 90.000,E1 123.833} C_DIS
LIN {X 0.072,Y -512.090,Z 379.485,A 0.000,B 0.000,C 90.000,E1 123.245} C_DIS
LIN {X -0.125,Y -509.245,Z 379.478,A 0.000,B 0.000,C 90.000,E1 122.084} C_DIS
LIN {X 0.110,Y -507.688,Z 379.475,A 0.000,B 0.000,C 90.000,E1 121.465} C_DIS
LIN {X 0.271,Y -504.121,Z 379.468,A 0.000,B 0.000,C 90.000,E1 120.256} C_DIS
LIN {X -0.176,Y -501.082,Z 379.463,A 0.000,B 0.000,C 90.000,E1 119.411} C_DIS
LIN {X 0.076,Y -496.629,Z 379.457,A 0.000,B 0.000,C 90.000,E1 118.180} C_DIS
LIN {X 0.021,Y -492.316,Z 379.451,A 0.000,B 0.000,C 90.000,E1 117.129} C_DIS
LIN {X -0.089,Y -486.403,Z 379.443,A 0.000,B 0.000,C 90.000,E1 115.771} C_DIS
LIN {X -0.059,Y -482.195,Z 379.438,A 0.000,B 0.000,C 90.000,E1 114.847} C_DIS
LIN {X -0.111,Y -475.611,Z 379.430,A 0.000,B 0.000,C 90.000,E1 113.462} C_DIS
LIN {X 0.153,Y -468.679,Z 379.423,A 0.000,B 0.000,C 90.000,E1 112.025} C_DIS
LIN {X 0.111,Y -461.586,Z 379.415,A 0.000,B 0.000,C 90.000,E1 110.610} C_DIS
LIN {X 0.043,Y -457.384,Z 379.410,A 0.000,B 0.000,C 90.000,E1 109.758} C_DIS
LIN {X 0.004,Y -457.363,Z 379.410,A 0.000,B 0.000,C 90.000,E1 109.758} C_DIS
LIN {X 0.210,Y -465.824,Z 379.387,A 0.000,B 0.000,C 90.000,E1 105.662} C_DIS
LIN {X -0.069,Y -467.383,Z 379.384,A 0.000,B 0.000,C 90.000,E1 105.064} C_DIS
LIN {X 0.187,Y -468.025,Z 379.382,A 0.000,B 0.000,C 90.000,E1 104.717} C_DIS
LIN {X 0.165,Y -476.237,Z 379.356,A 0.000,B 0.000,C 90.000,E1 100.018} C_DIS
LIN {X -0.049,Y -482.131,Z 379.330,A 0.000,B 0.000,C 90.000,E1 95.391} C_DIS
LIN {X 0.185,Y -485.529,Z 379.304,A 0.000,B 0.000,C 90.000,E1 90.745} C_DIS
LIN {X 0.218,Y -486.379,Z 379.280,A 0.000,B 0.000,C 90.000,E1 86.445} C_DIS
LIN {X 0.043,Y -486.350,Z 379.279,A 0.000,B 0.000,C 90.000,E1 86.159} C_DIS
LIN {X 0.121,Y -484.664,Z 379.253,A 0.000,B 0.000,C 90.000,E1 81.546} C_DIS
LIN {X 0.010,Y -480.583,Z 379.227,A 0.000,B 0.000,C 90.000,E1 76.937} C_DIS
LIN {X 0.189,Y -479.659,Z 379.224,A 0.000,B 0.000,C 90.000,E1 76.297} C_DIS
LIN {X 0.113,Y -474.270,Z 379.201,A 0.000,B 0.000,C 90.000,E1 72.181} C_DIS
LIN {X 0.073,Y -474.301,Z 379.201,A 0.000,B 0.000,C 90.000,E1 72.181} C_DIS
LIN {X -0.243,Y -483.568,Z 379.194,A 0.000,B 0.000,C 90.000,E1 70.913} C_DIS
LIN {X 0.242,Y -489.862,Z 379.189,A 0.000,B 0.000,C 90.000,E1 69.934} C_DIS
LIN {X 0.224,Y -498.041,Z 379.182,A 0.000,B 0.000,C 90.000,E1 68.720} C_DIS
LIN {X 0.151,Y -502.709,Z 379.178,A 0.000,B 0.000,C 90.000,E1 67.975} C_DIS
LIN {X -0.154,Y -506.172,Z 379.174,A 0.000,B 0.000,C 90.000,E1 67.411} C_DIS
LIN {X 0.227,Y -509.342,Z 379.171,A 0.000,B 0.000,C 90.000,E1 66.794} C_DIS
LIN {X -0.033,Y -512.519,Z 379.168,A 0.000,B 0.000,C 90.000,E1 66.230} C_DIS
LIN {X 0.027,Y -516.165,Z 379.164,A 0.000,B 0.000,C 90.000,E1 65.485} C_DIS
LIN {X 0.336,Y -519.357,Z 379.160,A 0.000,B 0.000,C 90.000,E1 64.717} C_DIS
LIN {X -0.182,Y -522.712,Z 379.155,A 0.000,B 0.000,C 90.000,E1 63.896} C_DIS
LIN {X -0.122,Y -524.801,Z 379.152,A 0.000,B 0.000,C 90.000,E1 63.307} C_DIS
LIN {X 0.117,Y -527.711,Z 379.147,A 0.000,B 0.000,C 90.000,E1 62.410} C_DIS
LIN {X -0.080,Y -530.478,Z 379.142,A 0.000,B 0.000,C 90.000,E1 61.563} C_DIS
LIN {X -0.106,Y -534.573,Z 379.134,A 0.000,B 0.000,C 90.000,E1 60.127} C_DIS
LIN {X 0.206,Y -538.397,Z 379.126,A 0.000,B 0.000,C 90.000,E1 58.663} C_DIS
LIN {X 0.114,Y -541.159,Z 379.120,A 0.000,B 0.000,C 90.000,E1 57.533} C_DIS
LIN {X -0.109,Y -543.687,Z 379.113,A 0.000,B 0.000,C 90.000,E1 56.421} C_DIS
LIN {X 0.126,Y -545.372,Z 379.109,A 0.000,B 0.000,C 90.000,E1 55.548} C_DIS
LIN {X 0.238,Y -546.798,Z 379.104,A 0.000,B 0.000,C 90.000,E1 54.689} C_DIS
LIN {X 0.048,Y -547.919,Z 379.099,A 0.000,B 0.000,C 90.000,E1 53.863} C_DIS
LIN {X 0.140,Y -548.597,Z 379.096,A 0.000,B 0.000,C 90.000,E1 53.290} C_DIS
LIN {X -0.145,Y -549.343,Z 379.091,A 0.000,B 0.000,C 90.000,E1 52.477} C_DIS
LIN {X 0.014,Y -549.675,Z 379.087,A 0.000,B 0.000,C 90.000,E1 51.618} C_DIS
LIN {X -0.255,Y -549.740,Z 379.082,A 0.000,B 0.000,C 90.000,E1 50.803} C_DIS
LIN {X 0.250,Y -549.393,Z 379.077,A 0.000,B 0.000,C 90.000,E1 49.908} C_DIS
LIN {X -0.070,Y -549.104,Z 379.074,A 0.000,B 0.000,C 90.000,E1 49.380} C_DIS
LIN {X 0.057,Y -548.056,Z 379.068,A 0.000,B 0.000,C 90.000,E1 48.243} C_DIS
LIN {X 0.130,Y -547.006,Z 379.063,A 0.000,B 0.000,C 90.000,E1 47.391} C_DIS
LIN {X 0.215,Y -544.984,Z 379.056,A 0.000,B 0.000,C 90.000,E1 45.972} C_DIS
LIN {X -0.118,Y -542.115,Z 379.045,A 0.000,B 0.000,C 90.000,E1 44.028} C_DIS
LIN {X -0.109,Y -539.764,Z 379.035,A 0.000,B 0.000,C 90.000,E1 42.324} C_DIS
LIN {X 0.209,Y -536.781,Z 379.022,A 0.000,B 0.000,C 90.000,E1 40.011} C_DIS
LIN {X 0.149,Y -534.187,Z 379.011,A 0.000,B 0.000,C 90.000,E1 38.016} C_DIS
LIN {X 0.133,Y -532.339,Z 379.003,A 0.000,B 0.000,C 90.000,E1 36.583} C_DIS
LIN {X -0.241,Y -530.007,Z 378.994,A 0.000,B 0.000,C 90.000,E1 34.898} C_DIS
LIN {X 0.091,Y -528.127,Z 378.986,A 0.000,B 0.000,C 90.000,E1 33.420} C_DIS
LIN {X 0.212,Y -525.932,Z 378.976,A 0.000,B 0.000,C 90.000,E1 31.671} C_DIS
LIN {X 0.104,Y -523.042,Z 378.963,A 0.000,B 0.000,C 90.000,E1 29.361} C_DIS
LIN {X -0.010,Y -520.674,Z 378.952,A 0.000,B 0.000,C 90.000,E1 27.334} C_DIS
LIN {X 0.032,Y -518.444,Z 378.941,A 0.000,B 0.000,C 90.000,E1 25.283} C_DIS
LIN {X -0.214,Y -516.378,Z 378.929,A 0.000,B 0.000,C 90.000,E1 23.259} C_DIS
LIN {X -0.068,Y -513.853,Z 378.913,A 0.000,B 0.000,C 90.000,E1 20.301} C_DIS
LIN {X 0.004,Y -512.061,Z 378.898,A 0.000,B 0.000,C 90.000,E1 17.638} C_DIS
LIN {X 0.206,Y -510.674,Z 378.883,A 0.000,B 0.000,C 90.000,E1 14.954} C_DIS
LIN {X 0.143,Y -509.905,Z 378.870,A 0.000,B 0.000,C 90.000,E1 12.591} C_DIS
LIN {X 0.218,Y -509.622,Z 378.852,A 0.000,B 0.000,C 90.000,E1 9.321} C_DIS
LIN {X 0.126,Y -510.024,Z 378.837,A 0.000,B 0.000,C 90.000,E1 6.663} C_DIS
LIN {X -0.010,Y -511.168,Z 378.822,A 0.000,B 0.000,C 90.000,E1 4.012} C_DIS
LIN {X -0.220,Y -513.048,Z 378.808,A 0.000,B 0.000,C 90.000,E1 1.375} C_DIS
LIN {X 0.234,Y -517.019,Z 378.787,A 0.000,B 0.000,C 90.000,E1 357.707} C_DIS
LIN {X -0.154,Y -519.989,Z 378.776,A 0.000,B 0.000,C 90.000,E1 355.698} C_DIS
LIN {X 0.028,Y -524.412,Z 378.761,A 0.000,B 0.000,C 90.000,E1 353.053} C_DIS
LIN {X 0.115,Y -532.748,Z 378.739,A 0.000,B 0.000,C 90.000,E1 348.993} C_DIS
LIN {X -0.004,Y -541.642,Z 378.720,A 0.000,B 0.000,C 90.000,E1 345.574} C_DIS
LIN {X 0.079,Y -546.464,Z 378.710,A 0.000,B 0.000,C 90.000,E1 343.866} C_DIS
LIN {X 0.132,Y -552.263,Z 378.700,A 0.000,B 0.000,C 90.000,E1 341.891} C_DIS
LIN {X -0.131,Y -557.202,Z 378.690,A 0.000,B 0.000,C 90.000,E1 340.242} C_DIS
LIN {X -0.282,Y -562.223,Z 378.681,A 0.000,B 0.000,C 90.000,E1 338.592} C_DIS
LIN {X -0.123,Y -567.206,Z 378.672,A 0.000,B 0.000,C 90.000,E1 336.922} C_DIS
LIN {X -0.151,Y -572.147,Z 378.663,A 0.000,B 0.000,C 90.000,E1 335.281} C_DIS
LIN {X 0.080,Y -576.351,Z 378.655,A 0.000,B 0.000,C 90.000,E1 333.896} C_DIS
LIN {X -0.153,Y -582.450,Z 378.645,A 0.000,B 0.000,C 90.000,E1 332.025} C_DIS
LIN {X 0.161,Y -587.818,Z 378.636,A 0.000,B 0.000,C 90.000,E1 330.383} C_DIS
LIN {X -0.117,Y -592.346,Z 378.628,A 0.000,B 0.000,C 90.000,E1 329.076} C_DIS
LIN {X -0.024,Y -596.890,Z 378.621,A 0.000,B 0.000,C 90.000,E1 327.740} C_DIS
LIN {X 0.118,Y -603.166,Z 378.611,A 0.000,B 0.000,C 90.000,E1 325.881} C_DIS
LIN {X 0.191,Y -610.659,Z 378.599,A 0.000,B 0.000,C 90.000,E1 323.783} C_DIS
LIN {X 0.031,Y -617.320,Z 378.589,A 0.000,B 0.000,C 90.000,E1 321.984} C_DIS
LIN {X -0.005,Y -620.239,Z 378.585,A 0.000,B 0.000,C 90.000,E1 321.215} C_DIS
LIN {X 0.262,Y -625.088,Z 378.577,A 0.000,B 0.000,C 90.000,E1 319.908} C_DIS
LIN {X -0.224,Y -628.857,Z 378.572,A 0.000,B 0.000,C 90.000,E1 318.933} C_DIS
LIN {X -0.007,Y -630.798,Z 378.569,A 0.000,B 0.000,C 90.000,E1 318.405} C_DIS
LIN {X -0.004,Y -634.470,Z 378.563,A 0.000,B 0.000,C 90.000,E1 317.391} C_DIS
LIN {X -0.139,Y -639.884,Z 378.555,A 0.000,B 0.000,C 90.000,E1 315.891} C_DIS
LIN {X 0.215,Y -646.326,Z 378.545,A 0.000,B 0.000,C 90.000,E1 314.109} C_DIS
LIN {X 0.321,Y -651.843,Z 378.537,A 0.000,B 0.000,C 90.000,E1 312.609} C_DIS
LIN {X 0.094,Y -657.323,Z 378.529,A 0.000,B 0.000,C 90.000,E1 311.148} C_DIS
LIN {X 0.022,Y -660.843,Z 378.523,A 0.000,B 0.000,C 90.000,E1 310.172} C_DIS
LIN {X -0.005,Y -664.335,Z 378.518,A 0.000,B 0.000,C 90.000,E1 309.197} C_DIS
LIN {X -0.343,Y -670.009,Z 378.508,A 0.000,B 0.000,C 90.000,E1 307.523} C_DIS
LIN {X 0.267,Y -673.128,Z 378.503,A 0.000,B 0.000,C 90.000,E1 306.503} C_DIS
LIN {X -0.425,Y -676.050,Z 378.498,A 0.000,B 0.000,C 90.000,E1 305.598} C_DIS
LIN {X -0.134,Y -678.835,Z 378.492,A 0.000,B 0.000,C 90.000,E1 304.612} C_DIS
LIN {X 0.197,Y -680.841,Z 378.488,A 0.000,B 0.000,C 90.000,E1 303.865} C_DIS
LIN {X -0.400,Y -683.290,Z 378.483,A 0.000,B 0.000,C 90.000,E1 302.959} C_DIS
LIN {X -0.220,Y -684.507,Z 378.480,A 0.000,B 0.000,C 90.000,E1 302.467} C_DIS
LIN {X 0.376,Y -686.766,Z 378.475,A 0.000,B 0.000,C 90.000,E1 301.465} C_DIS
LIN {X -0.156,Y -688.351,Z 378.471,A 0.000,B 0.000,C 90.000,E1 300.797} C_DIS
LIN {X -0.080,Y -689.711,Z 378.467,A 0.000,B 0.000,C 90.000,E1 300.079} C_DIS
LIN {X 0.355,Y -690.764,Z 378.463,A 0.000,B 0.000,C 90.000,E1 299.333} C_DIS
LIN {X -0.151,Y -691.500,Z 378.459,A 0.000,B 0.000,C 90.000,E1 298.665} C_DIS
LIN {X 0.086,Y -691.600,Z 378.458,A 0.000,B 0.000,C 90.000,E1 298.409} C_DIS
LIN {X -0.001,Y -691.884,Z 378.457,A 0.000,B 0.000,C 90.000,E1 298.180} C_DIS
LIN {X 0.116,Y -692.243,Z 378.453,A 0.000,B 0.000,C 90.000,E1 297.462} C_DIS
LIN {X 0.232,Y -692.385,Z 378.449,A 0.000,B 0.000,C 90.000,E1 296.744} C_DIS
LIN {X 0.038,Y -692.257,Z 378.445,A 0.000,B 0.000,C 90.000,E1 296.052} C_DIS
LIN {X 0.093,Y -691.725,Z 378.440,A 0.000,B 0.000,C 90.000,E1 295.103} C_DIS
LIN {X 0.142,Y -690.692,Z 378.434,A 0.000,B 0.000,C 90.000,E1 294.155} C_DIS
LIN {X -0.017,Y -690.093,Z 378.432,A 0.000,B 0.000,C 90.000,E1 293.695} C_DIS
LIN {X -0.052,Y -688.251,Z 378.425,A 0.000,B 0.000,C 90.000,E1 292.514} C_DIS
LIN {X 0.092,Y -686.939,Z 378.421,A 0.000,B 0.000,C 90.000,E1 291.791} C_DIS
LIN {X -0.028,Y -684.006,Z 378.413,A 0.000,B 0.000,C 90.000,E1 290.375} C_DIS
LIN {X -0.400,Y -681.595,Z 378.407,A 0.000,B 0.000,C 90.000,E1 289.214} C_DIS
LIN {X -0.173,Y -678.927,Z 378.400,A 0.000,B 0.000,C 90.000,E1 288.000} C_DIS
LIN {X -0.199,Y -676.333,Z 378.393,A 0.000,B 0.000,C 90.000,E1 286.804} C_DIS
LIN {X -0.376,Y -672.778,Z 378.384,A 0.000,B 0.000,C 90.000,E1 285.134} C_DIS
LIN {X 0.071,Y -666.727,Z 378.366,A 0.000,B 0.000,C 90.000,E1 281.951} C_DIS
LIN {X 0.069,Y -662.364,Z 378.350,A 0.000,B 0.000,C 90.000,E1 279.029} C_DIS
LIN {X 0.153,Y -659.201,Z 378.334,A 0.000,B 0.000,C 90.000,E1 276.087} C_DIS
LIN {X 0.216,Y -657.546,Z 378.319,A 0.000,B 0.000,C 90.000,E1 273.383} C_DIS
LIN {X 0.140,Y -656.851,Z 378.304,A 0.000,B 0.000,C 90.000,E1 270.688} C_DIS
LIN {X 0.312,Y -656.731,Z 378.296,A 0.000,B 0.000,C 90.000,E1 269.198} C_DIS
LIN {X 0.202,Y -656.880,Z 378.290,A 0.000,B 0.000,C 90.000,E1 268.224} C_DIS
LIN {X 0.029,Y -657.324,Z 378.279,A 0.000,B 0.000,C 90.000,E1 266.274} C_DIS
LIN {X -0.195,Y -657.675,Z 378.273,A 0.000,B 0.000,C 90.000,E1 265.065} C_DIS
LIN {X -0.276,Y -657.815,Z 378.267,A 0.000,B 0.000,C 90.000,E1 264.090} C_DIS
LIN {X 0.232,Y -657.507,Z 378.260,A 0.000,B 0.000,C 90.000,E1 262.818} C_DIS
LIN {X 0.211,Y -657.074,Z 378.255,A 0.000,B 0.000,C 90.000,E1 261.837} C_DIS
LIN {X -0.250,Y -656.513,Z 378.251,A 0.000,B 0.000,C 90.000,E1 261.141} C_DIS
LIN {X -0.066,Y -655.736,Z 378.247,A 0.000,B 0.000,C 90.000,E1 260.387} C_DIS
LIN {X -0.134,Y -654.116,Z 378.240,A 0.000,B 0.000,C 90.000,E1 259.162} C_DIS
LIN {X -0.230,Y -652.236,Z 378.233,A 0.000,B 0.000,C 90.000,E1 257.937} C_DIS
LIN {X 0.032,Y -651.057,Z 378.229,A 0.000,B 0.000,C 90.000,E1 257.173} C_DIS
LIN {X 0.283,Y -649.684,Z 378.225,A 0.000,B 0.000,C 90.000,E1 256.408} C_DIS
LIN {X 0.021,Y -648.703,Z 378.222,A 0.000,B 0.000,C 90.000,E1 255.936} C_DIS
LIN {X 0.104,Y -646.333,Z 378.216,A 0.000,B 0.000,C 90.000,E1 254.936} C_DIS
LIN {X -0.008,Y -645.093,Z 378.214,A 0.000,B 0.000,C 90.000,E1 254.448} C_DIS
LIN {X -0.298,Y -643.764,Z 378.211,A 0.000,B 0.000,C 90.000,E1 253.976} C_DIS
LIN {X 0.047,Y -641.533,Z 378.207,A 0.000,B 0.000,C 90.000,E1 253.196} C_DIS
LIN {X 0.032,Y -637.429,Z 378.200,A 0.000,B 0.000,C 90.000,E1 251.945} C_DIS
LIN {X -0.299,Y -634.825,Z 378.196,A 0.000,B 0.000,C 90.000,E1 251.221} C_DIS
LIN {X -0.041,Y -631.059,Z 378.190,A 0.000,B 0.000,C 90.000,E1 250.188} C_DIS
LIN {X 0.161,Y -627.193,Z 378.184,A 0.000,B 0.000,C 90.000,E1 249.156} C_DIS
LIN {X -0.281,Y -622.103,Z 378.177,A 0.000,B 0.000,C 90.000,E1 247.922} C_DIS
LIN {X 0.007,Y -616.783,Z 378.170,A 0.000,B 0.000,C 90.000,E1 246.613} C_DIS
LIN {X -0.358,Y -611.385,Z 378.163,A 0.000,B 0.000,C 90.000,E1 245.357} C_DIS
LIN {X -0.050,Y -604.820,Z 378.154,A 0.000,B 0.000,C 90.000,E1 243.768} C_DIS
LIN {X -0.349,Y -599.359,Z 378.147,A 0.000,B 0.000,C 90.000,E1 242.487} C_DIS
LIN {X 0.162,Y -591.735,Z 378.137,A 0.000,B 0.000,C 90.000,E1 240.589} C_DIS
LIN {X 0.011,Y -582.323,Z 378.123,A 0.000,B 0.000,C 90.000,E1 238.201} C_DIS
LIN {X 0.348,Y -574.532,Z 378.111,A 0.000,B 0.000,C 90.000,E1 236.008} C_DIS
LIN {X 0.066,Y -568.972,Z 378.102,A 0.000,B 0.000,C 90.000,E1 234.402} C_DIS
LIN {X -0.110,Y -564.442,Z 378.095,A 0.000,B 0.000,C 90.000,E1 233.050} C_DIS
LIN {X 0.320,Y -560.730,Z 378.089,A 0.000,B 0.000,C 90.000,E1 231.904} C_DIS
LIN {X -0.018,Y -554.926,Z 378.079,A 0.000,B 0.000,C 90.000,E1 230.275} C_DIS
LIN {X -0.065,Y -548.383,Z 378.068,A 0.000,B 0.000,C 90.000,E1 228.324} C_DIS
LIN {X 0.055,Y -542.933,Z 378.059,A 0.000,B 0.000,C 90.000,E1 226.620} C_DIS
LIN {X 0.053,Y -538.429,Z 378.051,A 0.000,B 0.000,C 90.000,E1 225.202} C_DIS
LIN {X -0.047,Y -533.102,Z 378.042,A 0.000,B 0.000,C 90.000,E1 223.500} C_DIS
LIN {X 0.112,Y -527.792,Z 378.032,A 0.000,B 0.000,C 90.000,E1 221.757} C_DIS
LIN {X 0.142,Y -521.840,Z 378.021,A 0.000,B 0.000,C 90.000,E1 219.725} C_DIS
LIN {X -0.247,Y -516.921,Z 378.011,A 0.000,B 0.000,C 90.000,E1 218.016} C_DIS
LIN {X 0.066,Y -512.163,Z 378.001,A 0.000,B 0.000,C 90.000,E1 216.217} C_DIS
LIN {X -0.096,Y -506.120,Z 377.988,A 0.000,B 0.000,C 90.000,E1 213.865} C_DIS
LIN {X 0.287,Y -499.695,Z 377.973,A 0.000,B 0.000,C 90.000,E1 211.131} C_DIS
LIN {X -0.193,Y -494.844,Z 377.961,A 0.000,B 0.000,C 90.000,E1 209.077} C_DIS
LIN {X 0.060,Y -490.020,Z 377.950,A 0.000,B 0.000,C 90.000,E1 206.924} C_DIS
LIN {X -0.060,Y -486.452,Z 377.941,A 0.000,B 0.000,C 90.000,E1 205.412} C_DIS
LIN {X 0.187,Y -484.334,Z 377.936,A 0.000,B 0.000,C 90.000,E1 204.463} C_DIS
LIN {X -0.035,Y -480.620,Z 377.928,A 0.000,B 0.000,C 90.000,E1 202.950} C_DIS
LIN {X -0.060,Y -477.686,Z 377.921,A 0.000,B 0.000,C 90.000,E1 201.716} C_DIS
LIN {X 0.261,Y -473.336,Z 377.910,A 0.000,B 0.000,C 90.000,E1 199.812} C_DIS
LIN {X 0.114,Y -468.382,Z 377.898,A 0.000,B 0.000,C 90.000,E1 197.638} C_DIS
LIN {X -0.222,Y -464.470,Z 377.888,A 0.000,B 0.000,C 90.000,E1 195.788} C_DIS
LIN {X 0.035,Y -460.147,Z 377.875,A 0.000,B 0.000,C 90.000,E1 193.536} C_DIS
LIN {X -0.041,Y -457.148,Z 377.866,A 0.000,B 0.000,C 90.000,E1 191.951} C_DIS
LIN {X -0.197,Y -453.290,Z 377.854,A 0.000,B 0.000,C 90.000,E1 189.726} C_DIS
LIN {X -0.176,Y -449.620,Z 377.841,A 0.000,B 0.000,C 90.000,E1 187.466} C_DIS
LIN {X 0.081,Y -446.297,Z 377.829,A 0.000,B 0.000,C 90.000,E1 185.163} C_DIS
LIN {X -0.220,Y -441.025,Z 377.803,A 0.000,B 0.000,C 90.000,E1 180.630} C_DIS
LIN {X 0.073,Y -438.632,Z 377.785,A 0.000,B 0.000,C 90.000,E1 177.306} C_DIS
LIN {X 0.037,Y -437.263,Z 377.765,A 0.000,B 0.000,C 90.000,E1 173.685} C_DIS
LIN {X -0.147,Y -437.425,Z 377.737,A 0.000,B 0.000,C 90.000,E1 168.757} C_DIS
LIN {X 0.143,Y -440.625,Z 377.708,A 0.000,B 0.000,C 90.000,E1 163.449} C_DIS
LIN {X -0.089,Y -442.558,Z 377.697,A 0.000,B 0.000,C 90.000,E1 161.511} C_DIS
LIN {X -0.129,Y -445.678,Z 377.683,A 0.000,B 0.000,C 90.000,E1 158.901} C_DIS
LIN {X -0.173,Y -449.547,Z 377.668,A 0.000,B 0.000,C 90.000,E1 156.305} C_DIS
LIN {X 0.123,Y -451.699,Z 377.661,A 0.000,B 0.000,C 90.000,E1 154.973} C_DIS
LIN {X -0.093,Y -457.180,Z 377.645,A 0.000,B 0.000,C 90.000,E1 152.103} C_DIS
LIN {X -0.094,Y -465.980,Z 377.624,A 0.000,B 0.000,C 90.000,E1 148.280} C_DIS
LIN {X -0.201,Y -472.091,Z 377.612,A 0.000,B 0.000,C 90.000,E1 146.087} C_DIS
LIN {X -0.076,Y -479.866,Z 377.598,A 0.000,B 0.000,C 90.000,E1 143.577} C_DIS
LIN {X -0.056,Y -485.048,Z 377.589,A 0.000,B 0.000,C 90.000,E1 142.029} C_DIS
LIN {X -0.087,Y -491.284,Z 377.579,A 0.000,B 0.000,C 90.000,E1 140.194} C_DIS
LIN {X -0.071,Y -495.396,Z 377.572,A 0.000,B 0.000,C 90.000,E1 138.976} C_DIS
LIN {X 0.010,Y -499.379,Z 377.565,A 0.000,B 0.000,C 90.000,E1 137.757} C_DIS
LIN {X 0.143,Y -503.102,Z 377.559,A 0.000,B 0.000,C 90.000,E1 136.539} C_DIS
LIN {X 0.084,Y -505.743,Z 377.554,A 0.000,B 0.000,C 90.000,E1 135.648} C_DIS
LIN {X 0.295,Y -508.943,Z 377.547,A 0.000,B 0.000,C 90.000,E1 134.433} C_DIS
LIN {X -0.050,Y -511.088,Z 377.542,A 0.000,B 0.000,C 90.000,E1 133.581} C_DIS
LIN {X -0.020,Y -513.033,Z 377.537,A 0.000,B 0.000,C 90.000,E1 132.690} C_DIS
LIN {X -0.062,Y -515.197,Z 377.531,A 0.000,B 0.000,C 90.000,E1 131.515} C_DIS
LIN {X 0.046,Y -516.546,Z 377.526,A 0.000,B 0.000,C 90.000,E1 130.620} C_DIS
LIN {X 0.172,Y -517.552,Z 377.521,A 0.000,B 0.000,C 90.000,E1 129.725} C_DIS
LIN {X 0.045,Y -517.971,Z 377.518,A 0.000,B 0.000,C 90.000,E1 129.152} C_DIS
LIN {X 0.249,Y -518.216,Z 377.514,A 0.000,B 0.000,C 90.000,E1 128.543} C_DIS
LIN {X 0.130,Y -518.178,Z 377.511,A 0.000,B 0.000,C 90.000,E1 127.971} C_DIS
LIN {X 0.269,Y -517.873,Z 377.506,A 0.000,B 0.000,C 90.000,E1 127.076} C_DIS
LIN {X 0.086,Y -517.205,Z 377.501,A 0.000,B 0.000,C 90.000,E1 126.217} C_DIS
LIN {X -0.106,Y -516.203,Z 377.496,A 0.000,B 0.000,C 90.000,E1 125.358} C_DIS
LIN {X -0.181,Y -514.908,Z 377.492,A 0.000,B 0.000,C 90.000,E1 124.485} C_DIS
LIN {X 0.026,Y -513.326,Z 377.487,A 0.000,B 0.000,C 90.000,E1 123.579} C_DIS
LIN {X -0.135,Y -512.122,Z 377.483,A 0.000,B 0.000,C 90.000,E1 123.007} C_DIS
LIN {X 0.187,Y -510.049,Z 377.478,A 0.000,B 0.000,C 90.000,E1 122.084} C_DIS
LIN {X 0.061,Y -507.684,Z 377.473,A 0.000,B 0.000,C 90.000,E1 121.209} C_DIS
LIN {X -0.092,Y -505.064,Z 377.469,A 0.000,B 0.000,C 90.000,E1 120.335} C_DIS
LIN {X 0.025,Y -501.168,Z 377.462,A 0.000,B 0.000,C 90.000,E1 119.127} C_DIS
LIN {X 0.270,Y -496.711,Z 377.455,A 0.000,B 0.000,C 90.000,E1 117.897} C_DIS
LIN {X -0.015,Y -492.452,Z 377.449,A 0.000,B 0.000,C 90.000,E1 116.873} C_DIS
LIN {X -0.122,Y -486.608,Z 377.442,A 0.000,B 0.000,C 90.000,E1 115.515} C_DIS
LIN {X -0.089,Y -482.448,Z 377.437,A 0.000,B 0.000,C 90.000,E1 114.591} C_DIS
LIN {X 0.071,Y -475.179,Z 377.428,A 0.000,B 0.000,C 90.000,E1 113.025} C_DIS
LIN {X 0.079,Y -467.456,Z 377.419,A 0.000,B 0.000,C 90.000,E1 111.461} C_DIS
LIN {X 0.138,Y -457.801,Z 377.409,A 0.000,B 0.000,C 90.000,E1 109.504} C_DIS
LIN {X 0.098,Y -457.796,Z 377.408,A 0.000,B 0.000,C 90.000,E1 109.504} C_DIS
LIN {X 0.063,Y -466.443,Z 377.386,A 0.000,B 0.000,C 90.000,E1 105.426} C_DIS
LIN {X 0.239,Y -467.940,Z 377.382,A 0.000,B 0.000,C 90.000,E1 104.773} C_DIS
LIN {X 0.204,Y -476.157,Z 377.356,A 0.000,B 0.000,C 90.000,E1 100.074} C_DIS
LIN {X -0.065,Y -482.067,Z 377.330,A 0.000,B 0.000,C 90.000,E1 95.454} C_DIS
LIN {X 0.210,Y -485.493,Z 377.305,A 0.000,B 0.000,C 90.000,E1 90.802} C_DIS
LIN {X 0.242,Y -486.385,Z 377.281,A 0.000,B 0.000,C 90.000,E1 86.502} C_DIS
LIN {X 0.067,Y -486.363,Z 377.279,A 0.000,B 0.000,C 90.000,E1 86.216} C_DIS
LIN {X 0.150,Y -484.688,Z 377.254,A 0.000,B 0.000,C 90.000,E1 81.602} C_DIS
LIN {X 0.049,Y -480.615,Z 377.228,A 0.000,B 0.000,C 90.000,E1 76.992} C_DIS
LIN {X -0.092,Y -480.272,Z 377.226,A 0.000,B 0.000,C 90.000,E1 76.700} C_DIS
LIN {X 0.208,Y -474.463,Z 377.202,A 0.000,B 0.000,C 90.000,E1 72.362} C_DIS
LIN {X 0.167,Y -474.479,Z 377.202,A 0.000,B 0.000,C 90.000,E1 72.362} C_DIS
LIN {X -0.172,Y -484.566,Z 377.194,A 0.000,B 0.000,C 90.000,E1 70.967} C_DIS
LIN {X 0.191,Y -492.794,Z 377.187,A 0.000,B 0.000,C 90.000,E1 69.699} C_DIS
LIN {X 0.275,Y -496.710,Z 377.184,A 0.000,B 0.000,C 90.000,E1 69.082} C_DIS
LIN {X 0.007,Y -501.435,Z 377.180,A 0.000,B 0.000,C 90.000,E1 68.358} C_DIS
LIN {X -0.037,Y -505.709,Z 377.176,A 0.000,B 0.000,C 90.000,E1 67.614} C_DIS
LIN {X 0.144,Y -508.669,Z 377.172,A 0.000,B 0.000,C 90.000,E1 66.997} C_DIS
LIN {X 0.239,Y -510.792,Z 377.170,A 0.000,B 0.000,C 90.000,E1 66.613} C_DIS
LIN {X -0.124,Y -512.161,Z 377.169,A 0.000,B 0.000,C 90.000,E1 66.357} C_DIS
LIN {X -0.174,Y -514.124,Z 377.166,A 0.000,B 0.000,C 90.000,E1 65.973} C_DIS
LIN {X 0.057,Y -516.660,Z 377.163,A 0.000,B 0.000,C 90.000,E1 65.409} C_DIS
LIN {X 0.150,Y -519.725,Z 377.159,A 0.000,B 0.000,C 90.000,E1 64.665} C_DIS
LIN {X -0.041,Y -522.012,Z 377.156,A 0.000,B 0.000,C 90.000,E1 64.101} C_DIS
LIN {X 0.160,Y -525.027,Z 377.151,A 0.000,B 0.000,C 90.000,E1 63.204} C_DIS
LIN {X 0.334,Y -528.629,Z 377.145,A 0.000,B 0.000,C 90.000,E1 62.025} C_DIS
LIN {X -0.273,Y -530.442,Z 377.142,A 0.000,B 0.000,C 90.000,E1 61.513} C_DIS
LIN {X -0.041,Y -534.441,Z 377.134,A 0.000,B 0.000,C 90.000,E1 60.049} C_DIS
LIN {X -0.006,Y -538.238,Z 377.126,A 0.000,B 0.000,C 90.000,E1 58.614} C_DIS
LIN {X 0.182,Y -541.015,Z 377.119,A 0.000,B 0.000,C 90.000,E1 57.454} C_DIS
LIN {X -0.038,Y -543.612,Z 377.113,A 0.000,B 0.000,C 90.000,E1 56.342} C_DIS
LIN {X 0.199,Y -545.394,Z 377.108,A 0.000,B 0.000,C 90.000,E1 55.468} C_DIS
LIN {X -0.004,Y -546.895,Z 377.104,A 0.000,B 0.000,C 90.000,E1 54.642} C_DIS
LIN {X 0.172,Y -548.419,Z 377.097,A 0.000,B 0.000,C 90.000,E1 53.497} C_DIS
LIN {X -0.167,Y -549.003,Z 377.094,A 0.000,B 0.000,C 90.000,E1 52.970} C_DIS
LIN {X -0.062,Y -549.581,Z 377.091,A 0.000,B 0.000,C 90.000,E1 52.396} C_DIS
LIN {X 0.046,Y -549.892,Z 377.088,A 0.000,B 0.000,C 90.000,E1 51.823} C_DIS
LIN {X 0.209,Y -550.164,Z 377.083,A 0.000,B 0.000,C 90.000,E1 50.964} C_DIS
LIN {X -0.057,Y -550.065,Z 377.079,A 0.000,B 0.000,C 90.000,E1 50.150} C_DIS
LIN {X 0.033,Y -549.745,Z 377.074,A 0.000,B 0.000,C 90.000,E1 49.299} C_DIS
LIN {X 0.125,Y -549.080,Z 377.069,A 0.000,B 0.000,C 90.000,E1 48.447} C_DIS
LIN {X 0.250,Y -547.822,Z 377.063,A 0.000,B 0.000,C 90.000,E1 47.310} C_DIS
LIN {X -0.051,Y -546.230,Z 377.057,A 0.000,B 0.000,C 90.000,E1 46.215} C_DIS
LIN {X 0.039,Y -543.015,Z 377.044,A 0.000,B 0.000,C 90.000,E1 43.947} C_DIS
LIN {X 0.065,Y -540.622,Z 377.035,A 0.000,B 0.000,C 90.000,E1 42.243} C_DIS
LIN {X 0.050,Y -538.020,Z 377.024,A 0.000,B 0.000,C 90.000,E1 40.253} C_DIS
LIN {X 0.030,Y -535.408,Z 377.013,A 0.000,B 0.000,C 90.000,E1 38.257} C_DIS
LIN {X 0.042,Y -533.209,Z 377.003,A 0.000,B 0.000,C 90.000,E1 36.537} C_DIS
LIN {X 0.000,Y -530.866,Z 376.993,A 0.000,B 0.000,C 90.000,E1 34.818} C_DIS
LIN {X 0.053,Y -529.000,Z 376.985,A 0.000,B 0.000,C 90.000,E1 33.372} C_DIS
LIN {X -0.247,Y -526.821,Z 376.976,A 0.000,B 0.000,C 90.000,E1 31.671} C_DIS
LIN {X -0.152,Y -524.652,Z 376.966,A 0.000,B 0.000,C 90.000,E1 29.922} C_DIS
LIN {X 0.150,Y -522.942,Z 376.958,A 0.000,B 0.000,C 90.000,E1 28.437} C_DIS
LIN {X 0.110,Y -520.954,Z 376.948,A 0.000,B 0.000,C 90.000,E1 26.693} C_DIS
LIN {X 0.016,Y -519.101,Z 376.939,A 0.000,B 0.000,C 90.000,E1 24.951} C_DIS
LIN {X 0.046,Y -517.078,Z 376.927,A 0.000,B 0.000,C 90.000,E1 22.898} C_DIS
LIN {X 0.100,Y -514.854,Z 376.913,A 0.000,B 0.000,C 90.000,E1 20.248} C_DIS
LIN {X 0.214,Y -513.076,Z 376.898,A 0.000,B 0.000,C 90.000,E1 17.583} C_DIS
LIN {X -0.074,Y -511.616,Z 376.881,A 0.000,B 0.000,C 90.000,E1 14.662} C_DIS
LIN {X -0.104,Y -510.920,Z 376.868,A 0.000,B 0.000,C 90.000,E1 12.299} C_DIS
LIN {X 0.050,Y -510.763,Z 376.852,A 0.000,B 0.000,C 90.000,E1 9.321} C_DIS
LIN {X 0.099,Y -511.147,Z 376.839,A 0.000,B 0.000,C 90.000,E1 6.947} C_DIS
LIN {X -0.099,Y -512.385,Z 376.822,A 0.000,B 0.000,C 90.000,E1 4.012} C_DIS
LIN {X 0.245,Y -514.332,Z 376.808,A 0.000,B 0.000,C 90.000,E1 1.318} C_DIS
LIN {X 0.206,Y -518.718,Z 376.786,A 0.000,B 0.000,C 90.000,E1 357.421} C_DIS
LIN {X -0.145,Y -521.761,Z 376.774,A 0.000,B 0.000,C 90.000,E1 355.412} C_DIS
LIN {X 0.151,Y -526.299,Z 376.760,A 0.000,B 0.000,C 90.000,E1 352.761} C_DIS
LIN {X -0.126,Y -535.504,Z 376.736,A 0.000,B 0.000,C 90.000,E1 348.465} C_DIS
LIN {X 0.110,Y -543.081,Z 376.720,A 0.000,B 0.000,C 90.000,E1 345.589} C_DIS
LIN {X -0.165,Y -547.915,Z 376.711,A 0.000,B 0.000,C 90.000,E1 343.921} C_DIS
LIN {X -0.071,Y -553.753,Z 376.700,A 0.000,B 0.000,C 90.000,E1 341.945} C_DIS
LIN {X 0.226,Y -558.716,Z 376.690,A 0.000,B 0.000,C 90.000,E1 340.242} C_DIS
LIN {X 0.111,Y -563.761,Z 376.681,A 0.000,B 0.000,C 90.000,E1 338.592} C_DIS
LIN {X -0.217,Y -568.762,Z 376.672,A 0.000,B 0.000,C 90.000,E1 336.975} C_DIS
LIN {X -0.089,Y -574.540,Z 376.661,A 0.000,B 0.000,C 90.000,E1 335.049} C_DIS
LIN {X 0.004,Y -581.373,Z 376.649,A 0.000,B 0.000,C 90.000,E1 332.871} C_DIS
LIN {X -0.114,Y -587.588,Z 376.639,A 0.000,B 0.000,C 90.000,E1 331.001} C_DIS
LIN {X -0.214,Y -593.004,Z 376.630,A 0.000,B 0.000,C 90.000,E1 329.410} C_DIS
LIN {X 0.111,Y -598.458,Z 376.621,A 0.000,B 0.000,C 90.000,E1 327.788} C_DIS
LIN {X -0.036,Y -604.707,Z 376.611,A 0.000,B 0.000,C 90.000,E1 325.960} C_DIS
LIN {X 0.074,Y -612.220,Z 376.599,A 0.000,B 0.000,C 90.000,E1 323.863} C_DIS
LIN {X -0.055,Y -618.889,Z 376.589,A 0.000,B 0.000,C 90.000,E1 322.065} C_DIS
LIN {X 0.028,Y -624.721,Z 376.581,A 0.000,B 0.000,C 90.000,E1 320.517} C_DIS
LIN {X -0.059,Y -628.480,Z 376.575,A 0.000,B 0.000,C 90.000,E1 319.504} C_DIS
LIN {X 0.097,Y -631.454,Z 376.571,A 0.000,B 0.000,C 90.000,E1 318.728} C_DIS
LIN {X -0.002,Y -636.026,Z 376.564,A 0.000,B 0.000,C 90.000,E1 317.472} C_DIS
LIN {X -0.106,Y -641.410,Z 376.555,A 0.000,B 0.000,C 90.000,E1 315.972} C_DIS
LIN {X 0.033,Y -645.063,Z 376.550,A 0.000,B 0.000,C 90.000,E1 314.960} C_DIS
END
